(* Logix 5000 project; controller ABB_Drive_Test vendor 1 type 14 code 149 rev 33.12; software revision 33.01; part 2 of 6 *)

        [6600] := 57, [6601] := 46, [6602] := 48, [6603] := 48, [6604] := 48, [6605] := 48, [6606] := 48, [6607] := 48, [6608] := 48, [6609] := 48, [6610] := 44, [6611] := 49, [6612] := 48, [6613] := 46, [6614] := 48, [6615] := 48, [6616] := 48, [6617] := 48, [6618] := 48, [6619] := 48, [6620] := 48, [6621] := 44, [6622] := 49, [6623] := 49, [6624] := 46, [6625] := 48, [6626] := 48, [6627] := 48, [6628] := 48, [6629] := 48, [6630] := 48, [6631] := 48, [6632] := 44, [6633] := 49, [6634] := 50, [6635] := 46, [6636] := 48, [6637] := 48, [6638] := 48, [6639] := 48, [6640] := 48, [6641] := 48, [6642] := 48, [6643] := 44, [6644] := 49, [6645] := 46, [6646] := 48, [6647] := 48, [6648] := 48, [6649] := 48, [6650] := 48, [6651] := 48, [6652] := 48, [6653] := 48, [6654] := 13, [6655] := 10, [6656] := 51, [6657] := 53, [6658] := 56, [6659] := 56,
        [6660] := 56, [6661] := 44, [6662] := 48, [6663] := 46, [6664] := 48, [6665] := 57, [6666] := 51, [6667] := 51, [6668] := 48, [6669] := 56, [6670] := 52, [6671] := 54, [6672] := 44, [6673] := 50, [6674] := 46, [6675] := 48, [6676] := 48, [6677] := 48, [6678] := 48, [6679] := 48, [6680] := 48, [6681] := 48, [6682] := 48, [6683] := 44, [6684] := 53, [6685] := 46, [6686] := 48, [6687] := 48, [6688] := 48, [6689] := 48, [6690] := 48, [6691] := 48, [6692] := 48, [6693] := 48, [6694] := 44, [6695] := 54, [6696] := 46, [6697] := 48, [6698] := 48, [6699] := 48, [6700] := 48, [6701] := 48, [6702] := 48, [6703] := 48, [6704] := 48, [6705] := 44, [6706] := 55, [6707] := 46, [6708] := 48, [6709] := 48, [6710] := 48, [6711] := 48, [6712] := 48, [6713] := 48, [6714] := 48, [6715] := 48, [6716] := 44, [6717] := 56, [6718] := 46, [6719] := 48,
        [6720] := 48, [6721] := 48, [6722] := 48, [6723] := 48, [6724] := 48, [6725] := 48, [6726] := 48, [6727] := 44, [6728] := 57, [6729] := 46, [6730] := 48, [6731] := 48, [6732] := 48, [6733] := 48, [6734] := 48, [6735] := 48, [6736] := 48, [6737] := 48, [6738] := 44, [6739] := 49, [6740] := 48, [6741] := 46, [6742] := 48, [6743] := 48, [6744] := 48, [6745] := 48, [6746] := 48, [6747] := 48, [6748] := 48, [6749] := 44, [6750] := 49, [6751] := 49, [6752] := 46, [6753] := 48, [6754] := 48, [6755] := 48, [6756] := 48, [6757] := 48, [6758] := 48, [6759] := 48, [6760] := 44, [6761] := 49, [6762] := 50, [6763] := 46, [6764] := 48, [6765] := 48, [6766] := 48, [6767] := 48, [6768] := 48, [6769] := 48, [6770] := 48, [6771] := 44, [6772] := 49, [6773] := 46, [6774] := 48, [6775] := 48, [6776] := 48, [6777] := 48, [6778] := 48, [6779] := 48,
        [6780] := 48, [6781] := 48, [6782] := 13, [6783] := 10, [6784] := 51, [6785] := 53, [6786] := 56, [6787] := 56, [6788] := 56, [6789] := 44, [6790] := 48, [6791] := 46, [6792] := 48, [6793] := 57, [6794] := 51, [6795] := 51, [6796] := 50, [6797] := 48, [6798] := 48, [6799] := 50, [6800] := 44, [6801] := 50, [6802] := 46, [6803] := 48, [6804] := 48, [6805] := 48, [6806] := 48, [6807] := 48, [6808] := 48, [6809] := 48, [6810] := 48, [6811] := 44, [6812] := 53, [6813] := 46, [6814] := 48, [6815] := 48, [6816] := 48, [6817] := 48, [6818] := 48, [6819] := 48, [6820] := 48, [6821] := 48, [6822] := 44, [6823] := 54, [6824] := 46, [6825] := 48, [6826] := 48, [6827] := 48, [6828] := 48, [6829] := 48, [6830] := 48, [6831] := 48, [6832] := 48, [6833] := 44, [6834] := 55, [6835] := 46, [6836] := 48, [6837] := 48, [6838] := 48, [6839] := 48,
        [6840] := 48, [6841] := 48, [6842] := 48, [6843] := 48, [6844] := 44, [6845] := 56, [6846] := 46, [6847] := 48, [6848] := 48, [6849] := 48, [6850] := 48, [6851] := 48, [6852] := 48, [6853] := 48, [6854] := 48, [6855] := 44, [6856] := 57, [6857] := 46, [6858] := 48, [6859] := 48, [6860] := 48, [6861] := 48, [6862] := 48, [6863] := 48, [6864] := 48, [6865] := 48, [6866] := 44, [6867] := 49, [6868] := 48, [6869] := 46, [6870] := 48, [6871] := 48, [6872] := 48, [6873] := 48, [6874] := 48, [6875] := 48, [6876] := 48, [6877] := 44, [6878] := 49, [6879] := 49, [6880] := 46, [6881] := 48, [6882] := 48, [6883] := 48, [6884] := 48, [6885] := 48, [6886] := 48, [6887] := 48, [6888] := 44, [6889] := 49, [6890] := 50, [6891] := 46, [6892] := 48, [6893] := 48, [6894] := 48, [6895] := 48, [6896] := 48, [6897] := 48, [6898] := 48, [6899] := 44,
        [6900] := 49, [6901] := 46, [6902] := 48, [6903] := 48, [6904] := 48, [6905] := 48, [6906] := 48, [6907] := 48, [6908] := 48, [6909] := 48, [6910] := 13, [6911] := 10, [6912] := 51, [6913] := 53, [6914] := 56, [6915] := 56, [6916] := 56, [6917] := 44, [6918] := 48, [6919] := 46, [6920] := 48, [6921] := 57, [6922] := 51, [6923] := 51, [6924] := 51, [6925] := 49, [6926] := 54, [6927] := 48, [6928] := 44, [6929] := 50, [6930] := 46, [6931] := 48, [6932] := 48, [6933] := 48, [6934] := 48, [6935] := 48, [6936] := 48, [6937] := 48, [6938] := 48, [6939] := 44, [6940] := 53, [6941] := 46, [6942] := 48, [6943] := 48, [6944] := 48, [6945] := 48, [6946] := 48, [6947] := 48, [6948] := 48, [6949] := 48, [6950] := 44, [6951] := 54, [6952] := 46, [6953] := 48, [6954] := 48, [6955] := 48, [6956] := 48, [6957] := 48, [6958] := 48, [6959] := 48,
        [6960] := 48, [6961] := 44, [6962] := 55, [6963] := 46, [6964] := 48, [6965] := 48, [6966] := 48, [6967] := 48, [6968] := 48, [6969] := 48, [6970] := 48, [6971] := 48, [6972] := 44, [6973] := 56, [6974] := 46, [6975] := 48, [6976] := 48, [6977] := 48, [6978] := 48, [6979] := 48, [6980] := 48, [6981] := 48, [6982] := 48, [6983] := 44, [6984] := 57, [6985] := 46, [6986] := 48, [6987] := 48, [6988] := 48, [6989] := 48, [6990] := 48, [6991] := 48, [6992] := 48, [6993] := 48, [6994] := 44, [6995] := 49, [6996] := 48, [6997] := 46, [6998] := 48, [6999] := 48, [7000] := 48, [7001] := 48, [7002] := 48, [7003] := 48, [7004] := 48, [7005] := 44, [7006] := 49, [7007] := 49, [7008] := 46, [7009] := 48, [7010] := 48, [7011] := 48, [7012] := 48, [7013] := 48, [7014] := 48, [7015] := 48, [7016] := 44, [7017] := 49, [7018] := 50, [7019] := 46,
        [7020] := 48, [7021] := 48, [7022] := 48, [7023] := 48, [7024] := 48, [7025] := 48, [7026] := 48, [7027] := 44, [7028] := 49, [7029] := 46, [7030] := 48, [7031] := 48, [7032] := 48, [7033] := 48, [7034] := 48, [7035] := 48, [7036] := 48, [7037] := 48, [7038] := 13, [7039] := 10, [7040] := 51, [7041] := 53, [7042] := 56, [7043] := 56, [7044] := 56, [7045] := 44, [7046] := 48, [7047] := 46, [7048] := 48, [7049] := 57, [7050] := 51, [7051] := 51, [7052] := 52, [7053] := 51, [7054] := 49, [7055] := 55, [7056] := 44, [7057] := 50, [7058] := 46, [7059] := 48, [7060] := 48, [7061] := 48, [7062] := 48, [7063] := 48, [7064] := 48, [7065] := 48, [7066] := 48, [7067] := 44, [7068] := 53, [7069] := 46, [7070] := 48, [7071] := 48, [7072] := 48, [7073] := 48, [7074] := 48, [7075] := 48, [7076] := 48, [7077] := 48, [7078] := 44, [7079] := 54,
        [7080] := 46, [7081] := 48, [7082] := 48, [7083] := 48, [7084] := 48, [7085] := 48, [7086] := 48, [7087] := 48, [7088] := 48, [7089] := 44, [7090] := 55, [7091] := 46, [7092] := 48, [7093] := 48, [7094] := 48, [7095] := 48, [7096] := 48, [7097] := 48, [7098] := 48, [7099] := 48, [7100] := 44, [7101] := 56, [7102] := 46, [7103] := 48, [7104] := 48, [7105] := 48, [7106] := 48, [7107] := 48, [7108] := 48, [7109] := 48, [7110] := 48, [7111] := 44, [7112] := 57, [7113] := 46, [7114] := 48, [7115] := 48, [7116] := 48, [7117] := 48, [7118] := 48, [7119] := 48, [7120] := 48, [7121] := 48, [7122] := 44, [7123] := 49, [7124] := 48, [7125] := 46, [7126] := 48, [7127] := 48, [7128] := 48, [7129] := 48, [7130] := 48, [7131] := 48, [7132] := 48, [7133] := 44, [7134] := 49, [7135] := 49, [7136] := 46, [7137] := 48, [7138] := 48, [7139] := 48,
        [7140] := 48, [7141] := 48, [7142] := 48, [7143] := 48, [7144] := 44, [7145] := 49, [7146] := 50, [7147] := 46, [7148] := 48, [7149] := 48, [7150] := 48, [7151] := 48, [7152] := 48, [7153] := 48, [7154] := 48, [7155] := 44, [7156] := 49, [7157] := 46, [7158] := 48, [7159] := 48, [7160] := 48, [7161] := 48, [7162] := 48, [7163] := 48, [7164] := 48, [7165] := 48, [7166] := 13, [7167] := 10, [7168] := 51, [7169] := 53, [7170] := 56, [7171] := 56, [7172] := 56, [7173] := 44, [7174] := 48, [7175] := 46, [7176] := 48, [7177] := 57, [7178] := 51, [7179] := 51, [7180] := 53, [7181] := 52, [7182] := 55, [7183] := 53, [7184] := 44, [7185] := 50, [7186] := 46, [7187] := 48, [7188] := 48, [7189] := 48, [7190] := 48, [7191] := 48, [7192] := 48, [7193] := 48, [7194] := 48, [7195] := 44, [7196] := 53, [7197] := 46, [7198] := 48, [7199] := 48,
        [7200] := 48, [7201] := 48, [7202] := 48, [7203] := 48, [7204] := 48, [7205] := 48, [7206] := 44, [7207] := 54, [7208] := 46, [7209] := 48, [7210] := 48, [7211] := 48, [7212] := 48, [7213] := 48, [7214] := 48, [7215] := 48, [7216] := 48, [7217] := 44, [7218] := 55, [7219] := 46, [7220] := 48, [7221] := 48, [7222] := 48, [7223] := 48, [7224] := 48, [7225] := 48, [7226] := 48, [7227] := 48, [7228] := 44, [7229] := 56, [7230] := 46, [7231] := 48, [7232] := 48, [7233] := 48, [7234] := 48, [7235] := 48, [7236] := 48, [7237] := 48, [7238] := 48, [7239] := 44, [7240] := 57, [7241] := 46, [7242] := 48, [7243] := 48, [7244] := 48, [7245] := 48, [7246] := 48, [7247] := 48, [7248] := 48, [7249] := 48, [7250] := 44, [7251] := 49, [7252] := 48, [7253] := 46, [7254] := 48, [7255] := 48, [7256] := 48, [7257] := 48, [7258] := 48, [7259] := 48,
        [7260] := 48, [7261] := 44, [7262] := 49, [7263] := 49, [7264] := 46, [7265] := 48, [7266] := 48, [7267] := 48, [7268] := 48, [7269] := 48, [7270] := 48, [7271] := 48, [7272] := 44, [7273] := 49, [7274] := 50, [7275] := 46, [7276] := 48, [7277] := 48, [7278] := 48, [7279] := 48, [7280] := 48, [7281] := 48, [7282] := 48, [7283] := 44, [7284] := 49, [7285] := 46, [7286] := 48, [7287] := 48, [7288] := 48, [7289] := 48, [7290] := 48, [7291] := 48, [7292] := 48, [7293] := 48, [7294] := 13, [7295] := 10, [7296] := 51, [7297] := 53, [7298] := 56, [7299] := 56, [7300] := 56, [7301] := 44, [7302] := 48, [7303] := 46, [7304] := 48, [7305] := 57, [7306] := 51, [7307] := 51, [7308] := 54, [7309] := 54, [7310] := 51, [7311] := 50, [7312] := 44, [7313] := 50, [7314] := 46, [7315] := 48, [7316] := 48, [7317] := 48, [7318] := 48, [7319] := 48,
        [7320] := 48, [7321] := 48, [7322] := 48, [7323] := 44, [7324] := 53, [7325] := 46, [7326] := 48, [7327] := 48, [7328] := 48, [7329] := 48, [7330] := 48, [7331] := 48, [7332] := 48, [7333] := 48, [7334] := 44, [7335] := 54, [7336] := 46, [7337] := 48, [7338] := 48, [7339] := 48, [7340] := 48, [7341] := 48, [7342] := 48, [7343] := 48, [7344] := 48, [7345] := 44, [7346] := 55, [7347] := 46, [7348] := 48, [7349] := 48, [7350] := 48, [7351] := 48, [7352] := 48, [7353] := 48, [7354] := 48, [7355] := 48, [7356] := 44, [7357] := 56, [7358] := 46, [7359] := 48, [7360] := 48, [7361] := 48, [7362] := 48, [7363] := 48, [7364] := 48, [7365] := 48, [7366] := 48, [7367] := 44, [7368] := 57, [7369] := 46, [7370] := 48, [7371] := 48, [7372] := 48, [7373] := 48, [7374] := 48, [7375] := 48, [7376] := 48, [7377] := 48, [7378] := 44, [7379] := 49,
        [7380] := 48, [7381] := 46, [7382] := 48, [7383] := 48, [7384] := 48, [7385] := 48, [7386] := 48, [7387] := 48, [7388] := 48, [7389] := 44, [7390] := 49, [7391] := 49, [7392] := 46, [7393] := 48, [7394] := 48, [7395] := 48, [7396] := 48, [7397] := 48, [7398] := 48, [7399] := 48, [7400] := 44, [7401] := 49, [7402] := 50, [7403] := 46, [7404] := 48, [7405] := 48, [7406] := 48, [7407] := 48, [7408] := 48, [7409] := 48, [7410] := 48, [7411] := 44, [7412] := 49, [7413] := 46, [7414] := 48, [7415] := 48, [7416] := 48, [7417] := 48, [7418] := 48, [7419] := 48, [7420] := 48, [7421] := 48, [7422] := 13, [7423] := 10, [7424] := 51, [7425] := 53, [7426] := 56, [7427] := 56, [7428] := 56, [7429] := 44, [7430] := 48, [7431] := 46, [7432] := 48, [7433] := 57, [7434] := 51, [7435] := 51, [7436] := 55, [7437] := 55, [7438] := 57, [7439] := 48,
        [7440] := 44, [7441] := 50, [7442] := 46, [7443] := 48, [7444] := 48, [7445] := 48, [7446] := 48, [7447] := 48, [7448] := 48, [7449] := 48, [7450] := 48, [7451] := 44, [7452] := 53, [7453] := 46, [7454] := 48, [7455] := 48, [7456] := 48, [7457] := 48, [7458] := 48, [7459] := 48, [7460] := 48, [7461] := 48, [7462] := 44, [7463] := 54, [7464] := 46, [7465] := 48, [7466] := 48, [7467] := 48, [7468] := 48, [7469] := 48, [7470] := 48, [7471] := 48, [7472] := 48, [7473] := 44, [7474] := 55, [7475] := 46, [7476] := 48, [7477] := 48, [7478] := 48, [7479] := 48, [7480] := 48, [7481] := 48, [7482] := 48, [7483] := 48, [7484] := 44, [7485] := 56, [7486] := 46, [7487] := 48, [7488] := 48, [7489] := 48, [7490] := 48, [7491] := 48, [7492] := 48, [7493] := 48, [7494] := 48, [7495] := 44, [7496] := 57, [7497] := 46, [7498] := 48, [7499] := 48,
        [7500] := 48, [7501] := 48, [7502] := 48, [7503] := 48, [7504] := 48, [7505] := 48, [7506] := 44, [7507] := 49, [7508] := 48, [7509] := 46, [7510] := 48, [7511] := 48, [7512] := 48, [7513] := 48, [7514] := 48, [7515] := 48, [7516] := 48, [7517] := 44, [7518] := 49, [7519] := 49, [7520] := 46, [7521] := 48, [7522] := 48, [7523] := 48, [7524] := 48, [7525] := 48, [7526] := 48, [7527] := 48, [7528] := 44, [7529] := 49, [7530] := 50, [7531] := 46, [7532] := 48, [7533] := 48, [7534] := 48, [7535] := 48, [7536] := 48, [7537] := 48, [7538] := 48, [7539] := 44, [7540] := 49, [7541] := 46, [7542] := 48, [7543] := 48, [7544] := 48, [7545] := 48, [7546] := 48, [7547] := 48, [7548] := 48, [7549] := 48, [7550] := 13, [7551] := 10, [7552] := 51, [7553] := 53, [7554] := 56, [7555] := 56, [7556] := 56, [7557] := 44, [7558] := 48, [7559] := 46,
        [7560] := 48, [7561] := 57, [7562] := 51, [7563] := 51, [7564] := 56, [7565] := 57, [7566] := 52, [7567] := 55, [7568] := 44, [7569] := 50, [7570] := 46, [7571] := 48, [7572] := 48, [7573] := 48, [7574] := 48, [7575] := 48, [7576] := 48, [7577] := 48, [7578] := 48, [7579] := 44, [7580] := 53, [7581] := 46, [7582] := 48, [7583] := 48, [7584] := 48, [7585] := 48, [7586] := 48, [7587] := 48, [7588] := 48, [7589] := 48, [7590] := 44, [7591] := 54, [7592] := 46, [7593] := 48, [7594] := 48, [7595] := 48, [7596] := 48, [7597] := 48, [7598] := 48, [7599] := 48, [7600] := 48, [7601] := 44, [7602] := 55, [7603] := 46, [7604] := 48, [7605] := 48, [7606] := 48, [7607] := 48, [7608] := 48, [7609] := 48, [7610] := 48, [7611] := 48, [7612] := 44, [7613] := 56, [7614] := 46, [7615] := 48, [7616] := 48, [7617] := 48, [7618] := 48, [7619] := 48,
        [7620] := 48, [7621] := 48, [7622] := 48, [7623] := 44, [7624] := 57, [7625] := 46, [7626] := 48, [7627] := 48, [7628] := 48, [7629] := 48, [7630] := 48, [7631] := 48, [7632] := 48, [7633] := 48, [7634] := 44, [7635] := 49, [7636] := 48, [7637] := 46, [7638] := 48, [7639] := 48, [7640] := 48, [7641] := 48, [7642] := 48, [7643] := 48, [7644] := 48, [7645] := 44, [7646] := 49, [7647] := 49, [7648] := 46, [7649] := 48, [7650] := 48, [7651] := 48, [7652] := 48, [7653] := 48, [7654] := 48, [7655] := 48, [7656] := 44, [7657] := 49, [7658] := 50, [7659] := 46, [7660] := 48, [7661] := 48, [7662] := 48, [7663] := 48, [7664] := 48, [7665] := 48, [7666] := 48, [7667] := 44, [7668] := 49, [7669] := 46, [7670] := 48, [7671] := 48, [7672] := 48, [7673] := 48, [7674] := 48, [7675] := 48, [7676] := 48, [7677] := 48, [7678] := 13, [7679] := 10,
        [7680] := 51, [7681] := 53, [7682] := 56, [7683] := 56, [7684] := 56, [7685] := 44, [7686] := 48, [7687] := 46, [7688] := 48, [7689] := 57, [7690] := 51, [7691] := 52, [7692] := 48, [7693] := 49, [7694] := 48, [7695] := 52, [7696] := 44, [7697] := 50, [7698] := 46, [7699] := 48, [7700] := 48, [7701] := 48, [7702] := 48, [7703] := 48, [7704] := 48, [7705] := 48, [7706] := 48, [7707] := 44, [7708] := 53, [7709] := 46, [7710] := 48, [7711] := 48, [7712] := 48, [7713] := 48, [7714] := 48, [7715] := 48, [7716] := 48, [7717] := 48, [7718] := 44, [7719] := 54, [7720] := 46, [7721] := 48, [7722] := 48, [7723] := 48, [7724] := 48, [7725] := 48, [7726] := 48, [7727] := 48, [7728] := 48, [7729] := 44, [7730] := 55, [7731] := 46, [7732] := 48, [7733] := 48, [7734] := 48, [7735] := 48, [7736] := 48, [7737] := 48, [7738] := 48, [7739] := 48,
        [7740] := 44, [7741] := 56, [7742] := 46, [7743] := 48, [7744] := 48, [7745] := 48, [7746] := 48, [7747] := 48, [7748] := 48, [7749] := 48, [7750] := 48, [7751] := 44, [7752] := 57, [7753] := 46, [7754] := 48, [7755] := 48, [7756] := 48, [7757] := 48, [7758] := 48, [7759] := 48, [7760] := 48, [7761] := 48, [7762] := 44, [7763] := 49, [7764] := 48, [7765] := 46, [7766] := 48, [7767] := 48, [7768] := 48, [7769] := 48, [7770] := 48, [7771] := 48, [7772] := 48, [7773] := 44, [7774] := 49, [7775] := 49, [7776] := 46, [7777] := 48, [7778] := 48, [7779] := 48, [7780] := 48, [7781] := 48, [7782] := 48, [7783] := 48, [7784] := 44, [7785] := 49, [7786] := 50, [7787] := 46, [7788] := 48, [7789] := 48, [7790] := 48, [7791] := 48, [7792] := 48, [7793] := 48, [7794] := 48, [7795] := 44, [7796] := 49, [7797] := 46, [7798] := 48, [7799] := 48,
        [7800] := 48, [7801] := 48, [7802] := 48, [7803] := 48, [7804] := 48, [7805] := 48, [7806] := 13, [7807] := 10, [7808] := 51, [7809] := 53, [7810] := 56, [7811] := 56, [7812] := 56, [7813] := 44, [7814] := 48, [7815] := 46, [7816] := 48, [7817] := 57, [7818] := 51, [7819] := 52, [7820] := 49, [7821] := 50, [7822] := 54, [7823] := 50, [7824] := 44, [7825] := 50, [7826] := 46, [7827] := 48, [7828] := 48, [7829] := 48, [7830] := 48, [7831] := 48, [7832] := 48, [7833] := 48, [7834] := 48, [7835] := 44, [7836] := 53, [7837] := 46, [7838] := 48, [7839] := 48, [7840] := 48, [7841] := 48, [7842] := 48, [7843] := 48, [7844] := 48, [7845] := 48, [7846] := 44, [7847] := 54, [7848] := 46, [7849] := 48, [7850] := 48, [7851] := 48, [7852] := 48, [7853] := 48, [7854] := 48, [7855] := 48, [7856] := 48, [7857] := 44, [7858] := 55, [7859] := 46,
        [7860] := 48, [7861] := 48, [7862] := 48, [7863] := 48, [7864] := 48, [7865] := 48, [7866] := 48, [7867] := 48, [7868] := 44, [7869] := 56, [7870] := 46, [7871] := 48, [7872] := 48, [7873] := 48, [7874] := 48, [7875] := 48, [7876] := 48, [7877] := 48, [7878] := 48, [7879] := 44, [7880] := 57, [7881] := 46, [7882] := 48, [7883] := 48, [7884] := 48, [7885] := 48, [7886] := 48, [7887] := 48, [7888] := 48, [7889] := 48, [7890] := 44, [7891] := 49, [7892] := 48, [7893] := 46, [7894] := 48, [7895] := 48, [7896] := 48, [7897] := 48, [7898] := 48, [7899] := 48, [7900] := 48, [7901] := 44, [7902] := 49, [7903] := 49, [7904] := 46, [7905] := 48, [7906] := 48, [7907] := 48, [7908] := 48, [7909] := 48, [7910] := 48, [7911] := 48, [7912] := 44, [7913] := 49, [7914] := 50, [7915] := 46, [7916] := 48, [7917] := 48, [7918] := 48, [7919] := 48,
        [7920] := 48, [7921] := 48, [7922] := 48, [7923] := 44, [7924] := 49, [7925] := 46, [7926] := 48, [7927] := 48, [7928] := 48, [7929] := 48, [7930] := 48, [7931] := 48, [7932] := 48, [7933] := 48, [7934] := 13, [7935] := 10, [7936] := 51, [7937] := 53, [7938] := 56, [7939] := 56, [7940] := 56, [7941] := 44, [7942] := 48, [7943] := 46, [7944] := 48, [7945] := 57, [7946] := 51, [7947] := 52, [7948] := 50, [7949] := 52, [7950] := 49, [7951] := 57, [7952] := 44, [7953] := 50, [7954] := 46, [7955] := 48, [7956] := 48, [7957] := 48, [7958] := 48, [7959] := 48, [7960] := 48, [7961] := 48, [7962] := 48, [7963] := 44, [7964] := 53, [7965] := 46, [7966] := 48, [7967] := 48, [7968] := 48, [7969] := 48, [7970] := 48, [7971] := 48, [7972] := 48, [7973] := 48, [7974] := 44, [7975] := 54, [7976] := 46, [7977] := 48, [7978] := 48, [7979] := 48,
        [7980] := 48, [7981] := 48, [7982] := 48, [7983] := 48, [7984] := 48, [7985] := 44, [7986] := 55, [7987] := 46, [7988] := 48, [7989] := 48, [7990] := 48, [7991] := 48, [7992] := 48, [7993] := 48, [7994] := 48, [7995] := 48, [7996] := 44, [7997] := 56, [7998] := 46, [7999] := 48, [8000] := 48, [8001] := 48, [8002] := 48, [8003] := 48, [8004] := 48, [8005] := 48, [8006] := 48, [8007] := 44, [8008] := 57, [8009] := 46, [8010] := 48, [8011] := 48, [8012] := 48, [8013] := 48, [8014] := 48, [8015] := 48, [8016] := 48, [8017] := 48, [8018] := 44, [8019] := 49, [8020] := 48, [8021] := 46, [8022] := 48, [8023] := 48, [8024] := 48, [8025] := 48, [8026] := 48, [8027] := 48, [8028] := 48, [8029] := 44, [8030] := 49, [8031] := 49, [8032] := 46, [8033] := 48, [8034] := 48, [8035] := 48, [8036] := 48, [8037] := 48, [8038] := 48, [8039] := 48,
        [8040] := 44, [8041] := 49, [8042] := 50, [8043] := 46, [8044] := 48, [8045] := 48, [8046] := 48, [8047] := 48, [8048] := 48, [8049] := 48, [8050] := 48, [8051] := 44, [8052] := 49, [8053] := 46, [8054] := 48, [8055] := 48, [8056] := 48, [8057] := 48, [8058] := 48, [8059] := 48, [8060] := 48, [8061] := 48, [8062] := 13, [8063] := 10, [8064] := 51, [8065] := 53, [8066] := 56, [8067] := 56, [8068] := 56, [8069] := 44, [8070] := 48, [8071] := 46, [8072] := 48, [8073] := 57, [8074] := 51, [8075] := 52, [8076] := 51, [8077] := 53, [8078] := 55, [8079] := 55, [8080] := 44, [8081] := 50, [8082] := 46, [8083] := 48, [8084] := 48, [8085] := 48, [8086] := 48, [8087] := 48, [8088] := 48, [8089] := 48, [8090] := 48, [8091] := 44, [8092] := 53, [8093] := 46, [8094] := 48, [8095] := 48, [8096] := 48, [8097] := 48, [8098] := 48, [8099] := 48,
        [8100] := 48, [8101] := 48, [8102] := 44, [8103] := 54, [8104] := 46, [8105] := 48, [8106] := 48, [8107] := 48, [8108] := 48, [8109] := 48, [8110] := 48, [8111] := 48, [8112] := 48, [8113] := 44, [8114] := 55, [8115] := 46, [8116] := 48, [8117] := 48, [8118] := 48, [8119] := 48, [8120] := 48, [8121] := 48, [8122] := 48, [8123] := 48, [8124] := 44, [8125] := 56, [8126] := 46, [8127] := 48, [8128] := 48, [8129] := 48, [8130] := 48, [8131] := 48, [8132] := 48, [8133] := 48, [8134] := 48, [8135] := 44, [8136] := 57, [8137] := 46, [8138] := 48, [8139] := 48, [8140] := 48, [8141] := 48, [8142] := 48, [8143] := 48, [8144] := 48, [8145] := 48, [8146] := 44, [8147] := 49, [8148] := 48, [8149] := 46, [8150] := 48, [8151] := 48, [8152] := 48, [8153] := 48, [8154] := 48, [8155] := 48, [8156] := 48, [8157] := 44, [8158] := 49, [8159] := 49,
        [8160] := 46, [8161] := 48, [8162] := 48, [8163] := 48, [8164] := 48, [8165] := 48, [8166] := 48, [8167] := 48, [8168] := 44, [8169] := 49, [8170] := 50, [8171] := 46, [8172] := 48, [8173] := 48, [8174] := 48, [8175] := 48, [8176] := 48, [8177] := 48, [8178] := 48, [8179] := 44, [8180] := 49, [8181] := 46, [8182] := 48, [8183] := 48, [8184] := 48, [8185] := 48, [8186] := 48, [8187] := 48, [8188] := 48, [8189] := 48, [8190] := 13, [8191] := 10, [8192] := 51, [8193] := 53, [8194] := 56, [8195] := 56, [8196] := 56, [8197] := 44, [8198] := 48, [8199] := 46, [8200] := 48, [8201] := 57, [8202] := 51, [8203] := 52, [8204] := 52, [8205] := 55, [8206] := 51, [8207] := 52, [8208] := 44, [8209] := 50, [8210] := 46, [8211] := 48, [8212] := 48, [8213] := 48, [8214] := 48, [8215] := 48, [8216] := 48, [8217] := 48, [8218] := 48, [8219] := 44,
        [8220] := 53, [8221] := 46, [8222] := 48, [8223] := 48, [8224] := 48, [8225] := 48, [8226] := 48, [8227] := 48, [8228] := 48, [8229] := 48, [8230] := 44, [8231] := 54, [8232] := 46, [8233] := 48, [8234] := 48, [8235] := 48, [8236] := 48, [8237] := 48, [8238] := 48, [8239] := 48, [8240] := 48, [8241] := 44, [8242] := 55, [8243] := 46, [8244] := 48, [8245] := 48, [8246] := 48, [8247] := 48, [8248] := 48, [8249] := 48, [8250] := 48, [8251] := 48, [8252] := 44, [8253] := 56, [8254] := 46, [8255] := 48, [8256] := 48, [8257] := 48, [8258] := 48, [8259] := 48, [8260] := 48, [8261] := 48, [8262] := 48, [8263] := 44, [8264] := 57, [8265] := 46, [8266] := 48, [8267] := 48, [8268] := 48, [8269] := 48, [8270] := 48, [8271] := 48, [8272] := 48, [8273] := 48, [8274] := 44, [8275] := 49, [8276] := 48, [8277] := 46, [8278] := 48, [8279] := 48,
        [8280] := 48, [8281] := 48, [8282] := 48, [8283] := 48, [8284] := 48, [8285] := 44, [8286] := 49, [8287] := 49, [8288] := 46, [8289] := 48, [8290] := 48, [8291] := 48, [8292] := 48, [8293] := 48, [8294] := 48, [8295] := 48, [8296] := 44, [8297] := 49, [8298] := 50, [8299] := 46, [8300] := 48, [8301] := 48, [8302] := 48, [8303] := 48, [8304] := 48, [8305] := 48, [8306] := 48, [8307] := 44, [8308] := 49, [8309] := 46, [8310] := 48, [8311] := 48, [8312] := 48, [8313] := 48, [8314] := 48, [8315] := 48, [8316] := 48, [8317] := 48, [8318] := 13, [8319] := 10, [8320] := 51, [8321] := 53, [8322] := 56, [8323] := 56, [8324] := 56, [8325] := 44, [8326] := 48, [8327] := 46, [8328] := 48, [8329] := 57, [8330] := 51, [8331] := 52, [8332] := 53, [8333] := 56, [8334] := 57, [8335] := 50, [8336] := 44, [8337] := 50, [8338] := 46, [8339] := 48,
        [8340] := 48, [8341] := 48, [8342] := 48, [8343] := 48, [8344] := 48, [8345] := 48, [8346] := 48, [8347] := 44, [8348] := 53, [8349] := 46, [8350] := 48, [8351] := 48, [8352] := 48, [8353] := 48, [8354] := 48, [8355] := 48, [8356] := 48, [8357] := 48, [8358] := 44, [8359] := 54, [8360] := 46, [8361] := 48, [8362] := 48, [8363] := 48, [8364] := 48, [8365] := 48, [8366] := 48, [8367] := 48, [8368] := 48, [8369] := 44, [8370] := 55, [8371] := 46, [8372] := 48, [8373] := 48, [8374] := 48, [8375] := 48, [8376] := 48, [8377] := 48, [8378] := 48, [8379] := 48, [8380] := 44, [8381] := 56, [8382] := 46, [8383] := 48, [8384] := 48, [8385] := 48, [8386] := 48, [8387] := 48, [8388] := 48, [8389] := 48, [8390] := 48, [8391] := 44, [8392] := 57, [8393] := 46, [8394] := 48, [8395] := 48, [8396] := 48, [8397] := 48, [8398] := 48, [8399] := 48,
        [8400] := 48, [8401] := 48, [8402] := 44, [8403] := 49, [8404] := 48, [8405] := 46, [8406] := 48, [8407] := 48, [8408] := 48, [8409] := 48, [8410] := 48, [8411] := 48, [8412] := 48, [8413] := 44, [8414] := 49, [8415] := 49, [8416] := 46, [8417] := 48, [8418] := 48, [8419] := 48, [8420] := 48, [8421] := 48, [8422] := 48, [8423] := 48, [8424] := 44, [8425] := 49, [8426] := 50, [8427] := 46, [8428] := 48, [8429] := 48, [8430] := 48, [8431] := 48, [8432] := 48, [8433] := 48, [8434] := 48, [8435] := 44, [8436] := 49, [8437] := 46, [8438] := 48, [8439] := 48, [8440] := 48, [8441] := 48, [8442] := 48, [8443] := 48, [8444] := 48, [8445] := 48, [8446] := 13, [8447] := 10, [8448] := 51, [8449] := 53, [8450] := 56, [8451] := 56, [8452] := 56, [8453] := 44, [8454] := 48, [8455] := 46, [8456] := 48, [8457] := 57, [8458] := 51, [8459] := 52,
        [8460] := 55, [8461] := 48, [8462] := 52, [8463] := 57, [8464] := 44, [8465] := 50, [8466] := 46, [8467] := 48, [8468] := 48, [8469] := 48, [8470] := 48, [8471] := 48, [8472] := 48, [8473] := 48, [8474] := 48, [8475] := 44, [8476] := 53, [8477] := 46, [8478] := 48, [8479] := 48, [8480] := 48, [8481] := 48, [8482] := 48, [8483] := 48, [8484] := 48, [8485] := 48, [8486] := 44, [8487] := 54, [8488] := 46, [8489] := 48, [8490] := 48, [8491] := 48, [8492] := 48, [8493] := 48, [8494] := 48, [8495] := 48, [8496] := 48, [8497] := 44, [8498] := 55, [8499] := 46, [8500] := 48, [8501] := 48, [8502] := 48, [8503] := 48, [8504] := 48, [8505] := 48, [8506] := 48, [8507] := 48, [8508] := 44, [8509] := 56, [8510] := 46, [8511] := 48, [8512] := 48, [8513] := 48, [8514] := 48, [8515] := 48, [8516] := 48, [8517] := 48, [8518] := 48, [8519] := 44,
        [8520] := 57, [8521] := 46, [8522] := 48, [8523] := 48, [8524] := 48, [8525] := 48, [8526] := 48, [8527] := 48, [8528] := 48, [8529] := 48, [8530] := 44, [8531] := 49, [8532] := 48, [8533] := 46, [8534] := 48, [8535] := 48, [8536] := 48, [8537] := 48, [8538] := 48, [8539] := 48, [8540] := 48, [8541] := 44, [8542] := 49, [8543] := 49, [8544] := 46, [8545] := 48, [8546] := 48, [8547] := 48, [8548] := 48, [8549] := 48, [8550] := 48, [8551] := 48, [8552] := 44, [8553] := 49, [8554] := 50, [8555] := 46, [8556] := 48, [8557] := 48, [8558] := 48, [8559] := 48, [8560] := 48, [8561] := 48, [8562] := 48, [8563] := 44, [8564] := 49, [8565] := 46, [8566] := 48, [8567] := 48, [8568] := 48, [8569] := 48, [8570] := 48, [8571] := 48, [8572] := 48, [8573] := 48, [8574] := 13, [8575] := 10, [8576] := 51, [8577] := 53, [8578] := 56, [8579] := 56,
        [8580] := 56, [8581] := 44, [8582] := 48, [8583] := 46, [8584] := 48, [8585] := 57, [8586] := 51, [8587] := 52, [8588] := 56, [8589] := 50, [8590] := 48, [8591] := 55, [8592] := 44, [8593] := 50, [8594] := 46, [8595] := 48, [8596] := 48, [8597] := 48, [8598] := 48, [8599] := 48, [8600] := 48, [8601] := 48, [8602] := 48, [8603] := 44, [8604] := 53, [8605] := 46, [8606] := 48, [8607] := 48, [8608] := 48, [8609] := 48, [8610] := 48, [8611] := 48, [8612] := 48, [8613] := 48, [8614] := 44, [8615] := 54, [8616] := 46, [8617] := 48, [8618] := 48, [8619] := 48, [8620] := 48, [8621] := 48, [8622] := 48, [8623] := 48, [8624] := 48, [8625] := 44, [8626] := 55, [8627] := 46, [8628] := 48, [8629] := 48, [8630] := 48, [8631] := 48, [8632] := 48, [8633] := 48, [8634] := 48, [8635] := 48, [8636] := 44, [8637] := 56, [8638] := 46, [8639] := 48,
        [8640] := 48, [8641] := 48, [8642] := 48, [8643] := 48, [8644] := 48, [8645] := 48, [8646] := 48, [8647] := 44, [8648] := 57, [8649] := 46, [8650] := 48, [8651] := 48, [8652] := 48, [8653] := 48, [8654] := 48, [8655] := 48, [8656] := 48, [8657] := 48, [8658] := 44, [8659] := 49, [8660] := 48, [8661] := 46, [8662] := 48, [8663] := 48, [8664] := 48, [8665] := 48, [8666] := 48, [8667] := 48, [8668] := 48, [8669] := 44, [8670] := 49, [8671] := 49, [8672] := 46, [8673] := 48, [8674] := 48, [8675] := 48, [8676] := 48, [8677] := 48, [8678] := 48, [8679] := 48, [8680] := 44, [8681] := 49, [8682] := 50, [8683] := 46, [8684] := 48, [8685] := 48, [8686] := 48, [8687] := 48, [8688] := 48, [8689] := 48, [8690] := 48, [8691] := 44, [8692] := 49, [8693] := 46, [8694] := 48, [8695] := 48, [8696] := 48, [8697] := 48, [8698] := 48, [8699] := 48,
        [8700] := 48, [8701] := 48, [8702] := 13, [8703] := 10, [8704] := 51, [8705] := 53, [8706] := 56, [8707] := 56, [8708] := 56, [8709] := 44, [8710] := 48, [8711] := 46, [8712] := 48, [8713] := 57, [8714] := 51, [8715] := 52, [8716] := 57, [8717] := 51, [8718] := 54, [8719] := 51, [8720] := 44, [8721] := 50, [8722] := 46, [8723] := 48, [8724] := 48, [8725] := 48, [8726] := 48, [8727] := 48, [8728] := 48, [8729] := 48, [8730] := 48, [8731] := 44, [8732] := 53, [8733] := 46, [8734] := 48, [8735] := 48, [8736] := 48, [8737] := 48, [8738] := 48, [8739] := 48, [8740] := 48, [8741] := 48, [8742] := 44, [8743] := 54, [8744] := 46, [8745] := 48, [8746] := 48, [8747] := 48, [8748] := 48, [8749] := 48, [8750] := 48, [8751] := 48, [8752] := 48, [8753] := 44, [8754] := 55, [8755] := 46, [8756] := 48, [8757] := 48, [8758] := 48, [8759] := 48,
        [8760] := 48, [8761] := 48, [8762] := 48, [8763] := 48, [8764] := 44, [8765] := 56, [8766] := 46, [8767] := 48, [8768] := 48, [8769] := 48, [8770] := 48, [8771] := 48, [8772] := 48, [8773] := 48, [8774] := 48, [8775] := 44, [8776] := 57, [8777] := 46, [8778] := 48, [8779] := 48, [8780] := 48, [8781] := 48, [8782] := 48, [8783] := 48, [8784] := 48, [8785] := 48, [8786] := 44, [8787] := 49, [8788] := 48, [8789] := 46, [8790] := 48, [8791] := 48, [8792] := 48, [8793] := 48, [8794] := 48, [8795] := 48, [8796] := 48, [8797] := 44, [8798] := 49, [8799] := 49, [8800] := 46, [8801] := 48, [8802] := 48, [8803] := 48, [8804] := 48, [8805] := 48, [8806] := 48, [8807] := 48, [8808] := 44, [8809] := 49, [8810] := 50, [8811] := 46, [8812] := 48, [8813] := 48, [8814] := 48, [8815] := 48, [8816] := 48, [8817] := 48, [8818] := 48, [8819] := 44,
        [8820] := 49, [8821] := 46, [8822] := 48, [8823] := 48, [8824] := 48, [8825] := 48, [8826] := 48, [8827] := 48, [8828] := 48, [8829] := 48, [8830] := 13, [8831] := 10, [8832] := 51, [8833] := 53, [8834] := 56, [8835] := 56, [8836] := 56, [8837] := 44, [8838] := 48, [8839] := 46, [8840] := 48, [8841] := 57, [8842] := 51, [8843] := 53, [8844] := 48, [8845] := 53, [8846] := 50, [8847] := 49, [8848] := 44, [8849] := 50, [8850] := 46, [8851] := 48, [8852] := 48, [8853] := 48, [8854] := 48, [8855] := 48, [8856] := 48, [8857] := 48, [8858] := 48, [8859] := 44, [8860] := 53, [8861] := 46, [8862] := 48, [8863] := 48, [8864] := 48, [8865] := 48, [8866] := 48, [8867] := 48, [8868] := 48, [8869] := 48, [8870] := 44, [8871] := 54, [8872] := 46, [8873] := 48, [8874] := 48, [8875] := 48, [8876] := 48, [8877] := 48, [8878] := 48, [8879] := 48,
        [8880] := 48, [8881] := 44, [8882] := 55, [8883] := 46, [8884] := 48, [8885] := 48, [8886] := 48, [8887] := 48, [8888] := 48, [8889] := 48, [8890] := 48, [8891] := 48, [8892] := 44, [8893] := 56, [8894] := 46, [8895] := 48, [8896] := 48, [8897] := 48, [8898] := 48, [8899] := 48, [8900] := 48, [8901] := 48, [8902] := 48, [8903] := 44, [8904] := 57, [8905] := 46, [8906] := 48, [8907] := 48, [8908] := 48, [8909] := 48, [8910] := 48, [8911] := 48, [8912] := 48, [8913] := 48, [8914] := 44, [8915] := 49, [8916] := 48, [8917] := 46, [8918] := 48, [8919] := 48, [8920] := 48, [8921] := 48, [8922] := 48, [8923] := 48, [8924] := 48, [8925] := 44, [8926] := 49, [8927] := 49, [8928] := 46, [8929] := 48, [8930] := 48, [8931] := 48, [8932] := 48, [8933] := 48, [8934] := 48, [8935] := 48, [8936] := 44, [8937] := 49, [8938] := 50, [8939] := 46,
        [8940] := 48, [8941] := 48, [8942] := 48, [8943] := 48, [8944] := 48, [8945] := 48, [8946] := 48, [8947] := 44, [8948] := 49, [8949] := 46, [8950] := 48, [8951] := 48, [8952] := 48, [8953] := 48, [8954] := 48, [8955] := 48, [8956] := 48, [8957] := 48, [8958] := 13, [8959] := 10, [8960] := 51, [8961] := 53, [8962] := 56, [8963] := 56, [8964] := 56, [8965] := 44, [8966] := 48, [8967] := 46, [8968] := 48, [8969] := 57, [8970] := 51, [8971] := 53, [8972] := 49, [8973] := 54, [8974] := 55, [8975] := 57, [8976] := 44, [8977] := 50, [8978] := 46, [8979] := 48, [8980] := 48, [8981] := 48, [8982] := 48, [8983] := 48, [8984] := 48, [8985] := 48, [8986] := 48, [8987] := 44, [8988] := 53, [8989] := 46, [8990] := 48, [8991] := 48, [8992] := 48, [8993] := 48, [8994] := 48, [8995] := 48, [8996] := 48, [8997] := 48, [8998] := 44, [8999] := 54,
        [9000] := 46, [9001] := 48, [9002] := 48, [9003] := 48, [9004] := 48, [9005] := 48, [9006] := 48, [9007] := 48, [9008] := 48, [9009] := 44, [9010] := 55, [9011] := 46, [9012] := 48, [9013] := 48, [9014] := 48, [9015] := 48, [9016] := 48, [9017] := 48, [9018] := 48, [9019] := 48, [9020] := 44, [9021] := 56, [9022] := 46, [9023] := 48, [9024] := 48, [9025] := 48, [9026] := 48, [9027] := 48, [9028] := 48, [9029] := 48, [9030] := 48, [9031] := 44, [9032] := 57, [9033] := 46, [9034] := 48, [9035] := 48, [9036] := 48, [9037] := 48, [9038] := 48, [9039] := 48, [9040] := 48, [9041] := 48, [9042] := 44, [9043] := 49, [9044] := 48, [9045] := 46, [9046] := 48, [9047] := 48, [9048] := 48, [9049] := 48, [9050] := 48, [9051] := 48, [9052] := 48, [9053] := 44, [9054] := 49, [9055] := 49, [9056] := 46, [9057] := 48, [9058] := 48, [9059] := 48,
        [9060] := 48, [9061] := 48, [9062] := 48, [9063] := 48, [9064] := 44, [9065] := 49, [9066] := 50, [9067] := 46, [9068] := 48, [9069] := 48, [9070] := 48, [9071] := 48, [9072] := 48, [9073] := 48, [9074] := 48, [9075] := 44, [9076] := 49, [9077] := 46, [9078] := 48, [9079] := 48, [9080] := 48, [9081] := 48, [9082] := 48, [9083] := 48, [9084] := 48, [9085] := 48, [9086] := 13, [9087] := 10, [9088] := 51, [9089] := 53, [9090] := 56, [9091] := 56, [9092] := 56, [9093] := 44, [9094] := 48, [9095] := 46, [9096] := 48, [9097] := 57, [9098] := 51, [9099] := 53, [9100] := 50, [9101] := 56, [9102] := 51, [9103] := 54, [9104] := 44, [9105] := 50, [9106] := 46, [9107] := 48, [9108] := 48, [9109] := 48, [9110] := 48, [9111] := 48, [9112] := 48, [9113] := 48, [9114] := 48, [9115] := 44, [9116] := 53, [9117] := 46, [9118] := 48, [9119] := 48,
        [9120] := 48, [9121] := 48, [9122] := 48, [9123] := 48, [9124] := 48, [9125] := 48, [9126] := 44, [9127] := 54, [9128] := 46, [9129] := 48, [9130] := 48, [9131] := 48, [9132] := 48, [9133] := 48, [9134] := 48, [9135] := 48, [9136] := 48, [9137] := 44, [9138] := 55, [9139] := 46, [9140] := 48, [9141] := 48, [9142] := 48, [9143] := 48, [9144] := 48, [9145] := 48, [9146] := 48, [9147] := 48, [9148] := 44, [9149] := 56, [9150] := 46, [9151] := 48, [9152] := 48, [9153] := 48, [9154] := 48, [9155] := 48, [9156] := 48, [9157] := 48, [9158] := 48, [9159] := 44, [9160] := 57, [9161] := 46, [9162] := 48, [9163] := 48, [9164] := 48, [9165] := 48, [9166] := 48, [9167] := 48, [9168] := 48, [9169] := 48, [9170] := 44, [9171] := 49, [9172] := 48, [9173] := 46, [9174] := 48, [9175] := 48, [9176] := 48, [9177] := 48, [9178] := 48, [9179] := 48,
        [9180] := 48, [9181] := 44, [9182] := 49, [9183] := 49, [9184] := 46, [9185] := 48, [9186] := 48, [9187] := 48, [9188] := 48, [9189] := 48, [9190] := 48, [9191] := 48, [9192] := 44, [9193] := 49, [9194] := 50, [9195] := 46, [9196] := 48, [9197] := 48, [9198] := 48, [9199] := 48, [9200] := 48, [9201] := 48, [9202] := 48, [9203] := 44, [9204] := 49, [9205] := 46, [9206] := 48, [9207] := 48, [9208] := 48, [9209] := 48, [9210] := 48, [9211] := 48, [9212] := 48, [9213] := 48, [9214] := 13, [9215] := 10, [9216] := 51, [9217] := 53, [9218] := 56, [9219] := 56, [9220] := 56, [9221] := 44, [9222] := 48, [9223] := 46, [9224] := 48, [9225] := 57, [9226] := 51, [9227] := 53, [9228] := 51, [9229] := 57, [9230] := 57, [9231] := 51, [9232] := 44, [9233] := 50, [9234] := 46, [9235] := 48, [9236] := 48, [9237] := 48, [9238] := 48, [9239] := 48,
        [9240] := 48, [9241] := 48, [9242] := 48, [9243] := 44, [9244] := 53, [9245] := 46, [9246] := 48, [9247] := 48, [9248] := 48, [9249] := 48, [9250] := 48, [9251] := 48, [9252] := 48, [9253] := 48, [9254] := 44, [9255] := 54, [9256] := 46, [9257] := 48, [9258] := 48, [9259] := 48, [9260] := 48, [9261] := 48, [9262] := 48, [9263] := 48, [9264] := 48, [9265] := 44, [9266] := 55, [9267] := 46, [9268] := 48, [9269] := 48, [9270] := 48, [9271] := 48, [9272] := 48, [9273] := 48, [9274] := 48, [9275] := 48, [9276] := 44, [9277] := 56, [9278] := 46, [9279] := 48, [9280] := 48, [9281] := 48, [9282] := 48, [9283] := 48, [9284] := 48, [9285] := 48, [9286] := 48, [9287] := 44, [9288] := 57, [9289] := 46, [9290] := 48, [9291] := 48, [9292] := 48, [9293] := 48, [9294] := 48, [9295] := 48, [9296] := 48, [9297] := 48, [9298] := 44, [9299] := 49,
        [9300] := 48, [9301] := 46, [9302] := 48, [9303] := 48, [9304] := 48, [9305] := 48, [9306] := 48, [9307] := 48, [9308] := 48, [9309] := 44, [9310] := 49, [9311] := 49, [9312] := 46, [9313] := 48, [9314] := 48, [9315] := 48, [9316] := 48, [9317] := 48, [9318] := 48, [9319] := 48, [9320] := 44, [9321] := 49, [9322] := 50, [9323] := 46, [9324] := 48, [9325] := 48, [9326] := 48, [9327] := 48, [9328] := 48, [9329] := 48, [9330] := 48, [9331] := 44, [9332] := 49, [9333] := 46, [9334] := 48, [9335] := 48, [9336] := 48, [9337] := 48, [9338] := 48, [9339] := 48, [9340] := 48, [9341] := 48, [9342] := 13, [9343] := 10, [9344] := 51, [9345] := 53, [9346] := 56, [9347] := 56, [9348] := 56, [9349] := 44, [9350] := 48, [9351] := 46, [9352] := 48, [9353] := 57, [9354] := 51, [9355] := 53, [9356] := 53, [9357] := 49, [9358] := 53, [9359] := 48,
        [9360] := 44, [9361] := 50, [9362] := 46, [9363] := 48, [9364] := 48, [9365] := 48, [9366] := 48, [9367] := 48, [9368] := 48, [9369] := 48, [9370] := 48, [9371] := 44, [9372] := 53, [9373] := 46, [9374] := 48, [9375] := 48, [9376] := 48, [9377] := 48, [9378] := 48, [9379] := 48, [9380] := 48, [9381] := 48, [9382] := 44, [9383] := 54, [9384] := 46, [9385] := 48, [9386] := 48, [9387] := 48, [9388] := 48, [9389] := 48, [9390] := 48, [9391] := 48, [9392] := 48, [9393] := 44, [9394] := 55, [9395] := 46, [9396] := 48, [9397] := 48, [9398] := 48, [9399] := 48, [9400] := 48, [9401] := 48, [9402] := 48, [9403] := 48, [9404] := 44, [9405] := 56, [9406] := 46, [9407] := 48, [9408] := 48, [9409] := 48, [9410] := 48, [9411] := 48, [9412] := 48, [9413] := 48, [9414] := 48, [9415] := 44, [9416] := 57, [9417] := 46, [9418] := 48, [9419] := 48,
        [9420] := 48, [9421] := 48, [9422] := 48, [9423] := 48, [9424] := 48, [9425] := 48, [9426] := 44, [9427] := 49, [9428] := 48, [9429] := 46, [9430] := 48, [9431] := 48, [9432] := 48, [9433] := 48, [9434] := 48, [9435] := 48, [9436] := 48, [9437] := 44, [9438] := 49, [9439] := 49, [9440] := 46, [9441] := 48, [9442] := 48, [9443] := 48, [9444] := 48, [9445] := 48, [9446] := 48, [9447] := 48, [9448] := 44, [9449] := 49, [9450] := 50, [9451] := 46, [9452] := 48, [9453] := 48, [9454] := 48, [9455] := 48, [9456] := 48, [9457] := 48, [9458] := 48, [9459] := 44, [9460] := 49, [9461] := 46, [9462] := 48, [9463] := 48, [9464] := 48, [9465] := 48, [9466] := 48, [9467] := 48, [9468] := 48, [9469] := 48, [9470] := 13, [9471] := 10, [9472] := 51, [9473] := 53, [9474] := 56, [9475] := 56, [9476] := 56, [9477] := 44, [9478] := 48, [9479] := 46,
        [9480] := 48, [9481] := 57, [9482] := 51, [9483] := 53, [9484] := 54, [9485] := 51, [9486] := 48, [9487] := 56, [9488] := 44, [9489] := 50, [9490] := 46, [9491] := 48, [9492] := 48, [9493] := 48, [9494] := 48, [9495] := 48, [9496] := 48, [9497] := 48, [9498] := 48, [9499] := 44, [9500] := 53, [9501] := 46, [9502] := 48, [9503] := 48, [9504] := 48, [9505] := 48, [9506] := 48, [9507] := 48, [9508] := 48, [9509] := 48, [9510] := 44, [9511] := 54, [9512] := 46, [9513] := 48, [9514] := 48, [9515] := 48, [9516] := 48, [9517] := 48, [9518] := 48, [9519] := 48, [9520] := 48, [9521] := 44, [9522] := 55, [9523] := 46, [9524] := 48, [9525] := 48, [9526] := 48, [9527] := 48, [9528] := 48, [9529] := 48, [9530] := 48, [9531] := 48, [9532] := 44, [9533] := 56, [9534] := 46, [9535] := 48, [9536] := 48, [9537] := 48, [9538] := 48, [9539] := 48,
        [9540] := 48, [9541] := 48, [9542] := 48, [9543] := 44, [9544] := 57, [9545] := 46, [9546] := 48, [9547] := 48, [9548] := 48, [9549] := 48, [9550] := 48, [9551] := 48, [9552] := 48, [9553] := 48, [9554] := 44, [9555] := 49, [9556] := 48, [9557] := 46, [9558] := 48, [9559] := 48, [9560] := 48, [9561] := 48, [9562] := 48, [9563] := 48, [9564] := 48, [9565] := 44, [9566] := 49, [9567] := 49, [9568] := 46, [9569] := 48, [9570] := 48, [9571] := 48, [9572] := 48, [9573] := 48, [9574] := 48, [9575] := 48, [9576] := 44, [9577] := 49, [9578] := 50, [9579] := 46, [9580] := 48, [9581] := 48, [9582] := 48, [9583] := 48, [9584] := 48, [9585] := 48, [9586] := 48, [9587] := 44, [9588] := 49, [9589] := 46, [9590] := 48, [9591] := 48, [9592] := 48, [9593] := 48, [9594] := 48, [9595] := 48, [9596] := 48, [9597] := 48, [9598] := 13, [9599] := 10,
        [9600] := 51, [9601] := 53, [9602] := 56, [9603] := 56, [9604] := 56, [9605] := 44, [9606] := 48, [9607] := 46, [9608] := 48, [9609] := 57, [9610] := 51, [9611] := 53, [9612] := 55, [9613] := 52, [9614] := 54, [9615] := 53, [9616] := 44, [9617] := 50, [9618] := 46, [9619] := 48, [9620] := 48, [9621] := 48, [9622] := 48, [9623] := 48, [9624] := 48, [9625] := 48, [9626] := 48, [9627] := 44, [9628] := 53, [9629] := 46, [9630] := 48, [9631] := 48, [9632] := 48, [9633] := 48, [9634] := 48, [9635] := 48, [9636] := 48, [9637] := 48, [9638] := 44, [9639] := 54, [9640] := 46, [9641] := 48, [9642] := 48, [9643] := 48, [9644] := 48, [9645] := 48, [9646] := 48, [9647] := 48, [9648] := 48, [9649] := 44, [9650] := 55, [9651] := 46, [9652] := 48, [9653] := 48, [9654] := 48, [9655] := 48, [9656] := 48, [9657] := 48, [9658] := 48, [9659] := 48,
        [9660] := 44, [9661] := 56, [9662] := 46, [9663] := 48, [9664] := 48, [9665] := 48, [9666] := 48, [9667] := 48, [9668] := 48, [9669] := 48, [9670] := 48, [9671] := 44, [9672] := 57, [9673] := 46, [9674] := 48, [9675] := 48, [9676] := 48, [9677] := 48, [9678] := 48, [9679] := 48, [9680] := 48, [9681] := 48, [9682] := 44, [9683] := 49, [9684] := 48, [9685] := 46, [9686] := 48, [9687] := 48, [9688] := 48, [9689] := 48, [9690] := 48, [9691] := 48, [9692] := 48, [9693] := 44, [9694] := 49, [9695] := 49, [9696] := 46, [9697] := 48, [9698] := 48, [9699] := 48, [9700] := 48, [9701] := 48, [9702] := 48, [9703] := 48, [9704] := 44, [9705] := 49, [9706] := 50, [9707] := 46, [9708] := 48, [9709] := 48, [9710] := 48, [9711] := 48, [9712] := 48, [9713] := 48, [9714] := 48, [9715] := 44, [9716] := 49, [9717] := 46, [9718] := 48, [9719] := 48,
        [9720] := 48, [9721] := 48, [9722] := 48, [9723] := 48, [9724] := 48, [9725] := 48, [9726] := 13, [9727] := 10, [9728] := 51, [9729] := 53, [9730] := 56, [9731] := 56, [9732] := 56, [9733] := 44, [9734] := 48, [9735] := 46, [9736] := 48, [9737] := 57, [9738] := 51, [9739] := 53, [9740] := 56, [9741] := 54, [9742] := 50, [9743] := 52, [9744] := 44, [9745] := 50, [9746] := 46, [9747] := 48, [9748] := 48, [9749] := 48, [9750] := 48, [9751] := 48, [9752] := 48, [9753] := 48, [9754] := 48, [9755] := 44, [9756] := 53, [9757] := 46, [9758] := 48, [9759] := 48, [9760] := 48, [9761] := 48, [9762] := 48, [9763] := 48, [9764] := 48, [9765] := 48, [9766] := 44, [9767] := 54, [9768] := 46, [9769] := 48, [9770] := 48, [9771] := 48, [9772] := 48, [9773] := 48, [9774] := 48, [9775] := 48, [9776] := 48, [9777] := 44, [9778] := 55, [9779] := 46,
        [9780] := 48, [9781] := 48, [9782] := 48, [9783] := 48, [9784] := 48, [9785] := 48, [9786] := 48, [9787] := 48, [9788] := 44, [9789] := 56, [9790] := 46, [9791] := 48, [9792] := 48, [9793] := 48, [9794] := 48, [9795] := 48, [9796] := 48, [9797] := 48, [9798] := 48, [9799] := 44, [9800] := 57, [9801] := 46, [9802] := 48, [9803] := 48, [9804] := 48, [9805] := 48, [9806] := 48, [9807] := 48, [9808] := 48, [9809] := 48, [9810] := 44, [9811] := 49, [9812] := 48, [9813] := 46, [9814] := 48, [9815] := 48, [9816] := 48, [9817] := 48, [9818] := 48, [9819] := 48, [9820] := 48, [9821] := 44, [9822] := 49, [9823] := 49, [9824] := 46, [9825] := 48, [9826] := 48, [9827] := 48, [9828] := 48, [9829] := 48, [9830] := 48, [9831] := 48, [9832] := 44, [9833] := 49, [9834] := 50, [9835] := 46, [9836] := 48, [9837] := 48, [9838] := 48, [9839] := 48,
        [9840] := 48, [9841] := 48, [9842] := 48, [9843] := 44, [9844] := 49, [9845] := 46, [9846] := 48, [9847] := 48, [9848] := 48, [9849] := 48, [9850] := 48, [9851] := 48, [9852] := 48, [9853] := 48, [9854] := 13, [9855] := 10, [9856] := 51, [9857] := 53, [9858] := 56, [9859] := 56, [9860] := 56, [9861] := 44, [9862] := 48, [9863] := 46, [9864] := 48, [9865] := 57, [9866] := 51, [9867] := 53, [9868] := 57, [9869] := 55, [9870] := 56, [9871] := 48, [9872] := 44, [9873] := 50, [9874] := 46, [9875] := 48, [9876] := 48, [9877] := 48, [9878] := 48, [9879] := 48, [9880] := 48, [9881] := 48, [9882] := 48, [9883] := 44, [9884] := 53, [9885] := 46, [9886] := 48, [9887] := 48, [9888] := 48, [9889] := 48, [9890] := 48, [9891] := 48, [9892] := 48, [9893] := 48, [9894] := 44, [9895] := 54, [9896] := 46, [9897] := 48, [9898] := 48, [9899] := 48,
        [9900] := 48, [9901] := 48, [9902] := 48, [9903] := 48, [9904] := 48, [9905] := 44, [9906] := 55, [9907] := 46, [9908] := 48, [9909] := 48, [9910] := 48, [9911] := 48, [9912] := 48, [9913] := 48, [9914] := 48, [9915] := 48, [9916] := 44, [9917] := 56, [9918] := 46, [9919] := 48, [9920] := 48, [9921] := 48, [9922] := 48, [9923] := 48, [9924] := 48, [9925] := 48, [9926] := 48, [9927] := 44, [9928] := 57, [9929] := 46, [9930] := 48, [9931] := 48, [9932] := 48, [9933] := 48, [9934] := 48, [9935] := 48, [9936] := 48, [9937] := 48, [9938] := 44, [9939] := 49, [9940] := 48, [9941] := 46, [9942] := 48, [9943] := 48, [9944] := 48, [9945] := 48, [9946] := 48, [9947] := 48, [9948] := 48, [9949] := 44, [9950] := 49, [9951] := 49, [9952] := 46, [9953] := 48, [9954] := 48, [9955] := 48, [9956] := 48, [9957] := 48, [9958] := 48, [9959] := 48,
        [9960] := 44, [9961] := 49, [9962] := 50, [9963] := 46, [9964] := 48, [9965] := 48, [9966] := 48, [9967] := 48, [9968] := 48, [9969] := 48, [9970] := 48, [9971] := 44, [9972] := 49, [9973] := 46, [9974] := 48, [9975] := 48, [9976] := 48, [9977] := 48, [9978] := 48, [9979] := 48, [9980] := 48, [9981] := 48, [9982] := 13, [9983] := 10, [9984] := 51, [9985] := 53, [9986] := 56, [9987] := 56, [9988] := 56, [9989] := 44, [9990] := 48, [9991] := 46, [9992] := 48, [9993] := 57, [9994] := 51, [9995] := 54, [9996] := 48, [9997] := 57, [9998] := 51, [9999] := 56, [10000] := 44, [10001] := 50, [10002] := 46, [10003] := 48, [10004] := 48, [10005] := 48, [10006] := 48, [10007] := 48, [10008] := 48, [10009] := 48, [10010] := 48, [10011] := 44, [10012] := 53, [10013] := 46, [10014] := 48, [10015] := 48, [10016] := 48, [10017] := 48, [10018] := 48, [10019] := 48,
        [10020] := 48, [10021] := 48, [10022] := 44, [10023] := 54, [10024] := 46, [10025] := 48, [10026] := 48, [10027] := 48, [10028] := 48, [10029] := 48, [10030] := 48, [10031] := 48, [10032] := 48, [10033] := 44, [10034] := 55, [10035] := 46, [10036] := 48, [10037] := 48, [10038] := 48, [10039] := 48, [10040] := 48, [10041] := 48, [10042] := 48, [10043] := 48, [10044] := 44, [10045] := 56, [10046] := 46, [10047] := 48, [10048] := 48, [10049] := 48, [10050] := 48, [10051] := 48, [10052] := 48, [10053] := 48, [10054] := 48, [10055] := 44, [10056] := 57, [10057] := 46, [10058] := 48, [10059] := 48, [10060] := 48, [10061] := 48, [10062] := 48, [10063] := 48, [10064] := 48, [10065] := 48, [10066] := 44, [10067] := 49, [10068] := 48, [10069] := 46, [10070] := 48, [10071] := 48, [10072] := 48, [10073] := 48, [10074] := 48, [10075] := 48, [10076] := 48, [10077] := 44, [10078] := 49, [10079] := 49,
        [10080] := 46, [10081] := 48, [10082] := 48, [10083] := 48, [10084] := 48, [10085] := 48, [10086] := 48, [10087] := 48, [10088] := 44, [10089] := 49, [10090] := 50, [10091] := 46, [10092] := 48, [10093] := 48, [10094] := 48, [10095] := 48, [10096] := 48, [10097] := 48, [10098] := 48, [10099] := 44, [10100] := 49, [10101] := 46, [10102] := 48, [10103] := 48, [10104] := 48, [10105] := 48, [10106] := 48, [10107] := 48, [10108] := 48, [10109] := 48, [10110] := 13, [10111] := 10, [10112] := 49, [10113] := 48, [10114] := 44, [10115] := 54, [10116] := 46, [10117] := 54, [10118] := 54, [10119] := 54, [10120] := 54, [10121] := 54, [10122] := 54, [10123] := 48, [10124] := 51, [10125] := 44, [10126] := 55, [10127] := 46, [10128] := 55, [10129] := 55, [10130] := 55, [10131] := 55, [10132] := 55, [10133] := 55, [10134] := 54, [10135] := 55, [10136] := 44, [10137] := 56, [10138] := 46, [10139] := 56,
        [10140] := 56, [10141] := 56, [10142] := 56, [10143] := 56, [10144] := 57, [10145] := 51, [10146] := 49, [10147] := 44, [10148] := 49, [10149] := 48, [10150] := 46, [10151] := 48, [10152] := 48, [10153] := 48, [10154] := 48, [10155] := 48, [10156] := 48, [10157] := 48, [10158] := 44, [10159] := 48, [10160] := 46, [10161] := 48, [10162] := 13, [10163] := 10, [10164] := 52, [10165] := 49, [10166] := 56, [10167] := 48, [10168] := 51, [10169] := 44, [10170] := 48, [10171] := 46, [10172] := 51, [10173] := 50, [10174] := 53, [10175] := 50, [10176] := 50, [10177] := 57, [10178] := 48, [10179] := 50, [10180] := 44, [10181] := 49, [10182] := 46, [10183] := 49, [10184] := 48, [10185] := 48, [10186] := 48, [10187] := 48, [10188] := 48, [10189] := 48, [10190] := 50, [10191] := 44, [10192] := 50, [10193] := 46, [10194] := 50, [10195] := 50, [10196] := 48, [10197] := 48, [10198] := 48, [10199] := 48,
        [10200] := 48, [10201] := 51, [10202] := 44, [10203] := 51, [10204] := 46, [10205] := 51, [10206] := 51, [10207] := 50, [10208] := 57, [10209] := 57, [10210] := 57, [10211] := 57, [10212] := 52, [10213] := 44, [10214] := 52, [10215] := 46, [10216] := 52, [10217] := 52, [10218] := 52, [10219] := 51, [10220] := 57, [10221] := 57, [10222] := 56, [10223] := 51, [10224] := 44, [10225] := 53, [10226] := 46, [10227] := 53, [10228] := 53, [10229] := 53, [10230] := 53, [10231] := 53, [10232] := 48, [10233] := 49, [10234] := 48, [10235] := 44, [10236] := 54, [10237] := 46, [10238] := 54, [10239] := 54, [10240] := 54, [10241] := 54, [10242] := 54, [10243] := 54, [10244] := 48, [10245] := 51, [10246] := 44, [10247] := 55, [10248] := 46, [10249] := 55, [10250] := 55, [10251] := 55, [10252] := 55, [10253] := 55, [10254] := 55, [10255] := 54, [10256] := 55, [10257] := 44, [10258] := 56, [10259] := 46,
        [10260] := 56, [10261] := 56, [10262] := 56, [10263] := 56, [10264] := 56, [10265] := 57, [10266] := 51, [10267] := 49, [10268] := 44, [10269] := 49, [10270] := 48, [10271] := 46, [10272] := 48, [10273] := 48, [10274] := 48, [10275] := 48, [10276] := 48, [10277] := 48, [10278] := 48, [10279] := 44, [10280] := 48, [10281] := 46, [10282] := 48, [10283] := 13, [10284] := 10, [10285] := 52, [10286] := 49, [10287] := 56, [10288] := 48, [10289] := 51, [10290] := 44, [10291] := 48, [10292] := 46, [10293] := 51, [10294] := 50, [10295] := 53, [10296] := 50, [10297] := 52, [10298] := 48, [10299] := 54, [10300] := 49, [10301] := 44, [10302] := 49, [10303] := 46, [10304] := 49, [10305] := 48, [10306] := 48, [10307] := 48, [10308] := 48, [10309] := 48, [10310] := 48, [10311] := 50, [10312] := 44, [10313] := 50, [10314] := 46, [10315] := 50, [10316] := 50, [10317] := 48, [10318] := 48, [10319] := 48,
        [10320] := 48, [10321] := 48, [10322] := 51, [10323] := 44, [10324] := 51, [10325] := 46, [10326] := 51, [10327] := 51, [10328] := 50, [10329] := 57, [10330] := 57, [10331] := 57, [10332] := 57, [10333] := 52, [10334] := 44, [10335] := 52, [10336] := 46, [10337] := 52, [10338] := 52, [10339] := 52, [10340] := 51, [10341] := 57, [10342] := 57, [10343] := 56, [10344] := 51, [10345] := 44, [10346] := 53, [10347] := 46, [10348] := 53, [10349] := 53, [10350] := 53, [10351] := 53, [10352] := 53, [10353] := 48, [10354] := 49, [10355] := 48, [10356] := 44, [10357] := 54, [10358] := 46, [10359] := 54, [10360] := 54, [10361] := 54, [10362] := 54, [10363] := 54, [10364] := 54, [10365] := 48, [10366] := 51, [10367] := 44, [10368] := 55, [10369] := 46, [10370] := 55, [10371] := 55, [10372] := 55, [10373] := 55, [10374] := 55, [10375] := 55, [10376] := 54, [10377] := 55, [10378] := 44, [10379] := 56,
        [10380] := 46, [10381] := 56, [10382] := 56, [10383] := 56, [10384] := 56, [10385] := 56, [10386] := 57, [10387] := 51, [10388] := 49, [10389] := 44, [10390] := 49, [10391] := 48, [10392] := 46, [10393] := 48, [10394] := 48, [10395] := 48, [10396] := 48, [10397] := 48, [10398] := 48, [10399] := 48, [10400] := 44, [10401] := 48, [10402] := 46, [10403] := 48, [10404] := 13, [10405] := 10, [10406] := 52, [10407] := 49, [10408] := 56, [10409] := 48, [10410] := 51, [10411] := 44, [10412] := 48, [10413] := 46, [10414] := 51, [10415] := 50, [10416] := 53, [10417] := 50, [10418] := 53, [10419] := 50, [10420] := 49, [10421] := 56, [10422] := 44, [10423] := 49, [10424] := 46, [10425] := 49, [10426] := 48, [10427] := 48, [10428] := 48, [10429] := 48, [10430] := 48, [10431] := 48, [10432] := 50, [10433] := 44, [10434] := 50, [10435] := 46, [10436] := 50, [10437] := 50, [10438] := 48, [10439] := 48,
        [10440] := 48, [10441] := 48, [10442] := 48, [10443] := 51, [10444] := 44, [10445] := 51, [10446] := 46, [10447] := 51, [10448] := 51, [10449] := 50, [10450] := 57, [10451] := 57, [10452] := 57, [10453] := 57, [10454] := 52, [10455] := 44, [10456] := 52, [10457] := 46, [10458] := 52, [10459] := 52, [10460] := 52, [10461] := 51, [10462] := 57, [10463] := 57, [10464] := 56, [10465] := 51, [10466] := 44, [10467] := 53, [10468] := 46, [10469] := 53, [10470] := 53, [10471] := 53, [10472] := 53, [10473] := 53, [10474] := 48, [10475] := 49, [10476] := 48, [10477] := 44, [10478] := 54, [10479] := 46, [10480] := 54, [10481] := 54, [10482] := 54, [10483] := 54, [10484] := 54, [10485] := 54, [10486] := 48, [10487] := 51, [10488] := 44, [10489] := 55, [10490] := 46, [10491] := 55, [10492] := 55, [10493] := 55, [10494] := 55, [10495] := 55, [10496] := 55, [10497] := 54, [10498] := 55, [10499] := 44,
        [10500] := 56, [10501] := 46, [10502] := 56, [10503] := 56, [10504] := 56, [10505] := 56, [10506] := 56, [10507] := 57, [10508] := 51, [10509] := 49, [10510] := 44, [10511] := 49, [10512] := 48, [10513] := 46, [10514] := 48, [10515] := 48, [10516] := 48, [10517] := 48, [10518] := 48, [10519] := 48, [10520] := 48, [10521] := 44, [10522] := 48, [10523] := 46, [10524] := 48, [10525] := 13, [10526] := 10, [10527] := 52, [10528] := 49, [10529] := 56, [10530] := 48, [10531] := 51, [10532] := 44, [10533] := 48, [10534] := 46, [10535] := 51, [10536] := 50, [10537] := 53, [10538] := 50, [10539] := 54, [10540] := 51, [10541] := 55, [10542] := 52, [10543] := 44, [10544] := 49, [10545] := 46, [10546] := 49, [10547] := 48, [10548] := 48, [10549] := 48, [10550] := 48, [10551] := 48, [10552] := 48, [10553] := 50, [10554] := 44, [10555] := 50, [10556] := 46, [10557] := 50, [10558] := 50, [10559] := 48,
        [10560] := 48, [10561] := 48, [10562] := 48, [10563] := 48, [10564] := 51, [10565] := 44, [10566] := 51, [10567] := 46, [10568] := 51, [10569] := 51, [10570] := 50, [10571] := 57, [10572] := 57, [10573] := 57, [10574] := 57, [10575] := 52, [10576] := 44, [10577] := 52, [10578] := 46, [10579] := 52, [10580] := 52, [10581] := 52, [10582] := 51, [10583] := 57, [10584] := 57, [10585] := 56, [10586] := 51, [10587] := 44, [10588] := 53, [10589] := 46, [10590] := 53, [10591] := 53, [10592] := 53, [10593] := 53, [10594] := 53, [10595] := 48, [10596] := 49, [10597] := 48, [10598] := 44, [10599] := 54, [10600] := 46, [10601] := 54, [10602] := 54, [10603] := 54, [10604] := 54, [10605] := 54, [10606] := 54, [10607] := 48, [10608] := 51, [10609] := 44, [10610] := 55, [10611] := 46, [10612] := 55, [10613] := 55, [10614] := 55, [10615] := 55, [10616] := 55, [10617] := 55, [10618] := 54, [10619] := 55,
        [10620] := 44, [10621] := 56, [10622] := 46, [10623] := 56, [10624] := 56, [10625] := 56, [10626] := 56, [10627] := 56, [10628] := 57, [10629] := 51, [10630] := 49, [10631] := 44, [10632] := 49, [10633] := 48, [10634] := 46, [10635] := 48, [10636] := 48, [10637] := 48, [10638] := 48, [10639] := 48, [10640] := 48, [10641] := 48, [10642] := 44, [10643] := 48, [10644] := 46, [10645] := 48, [10646] := 13, [10647] := 10, [10648] := 52, [10649] := 49, [10650] := 56, [10651] := 48, [10652] := 51, [10653] := 44, [10654] := 48, [10655] := 46, [10656] := 51, [10657] := 50, [10658] := 53, [10659] := 50, [10660] := 55, [10661] := 53, [10662] := 51, [10663] := 51, [10664] := 44, [10665] := 49, [10666] := 46, [10667] := 49, [10668] := 48, [10669] := 48, [10670] := 48, [10671] := 48, [10672] := 48, [10673] := 48, [10674] := 50, [10675] := 44, [10676] := 50, [10677] := 46, [10678] := 50, [10679] := 50,
        [10680] := 48, [10681] := 48, [10682] := 48, [10683] := 48, [10684] := 48, [10685] := 51, [10686] := 44, [10687] := 51, [10688] := 46, [10689] := 51, [10690] := 51, [10691] := 50, [10692] := 57, [10693] := 57, [10694] := 57, [10695] := 57, [10696] := 52, [10697] := 44, [10698] := 52, [10699] := 46, [10700] := 52, [10701] := 52, [10702] := 52, [10703] := 51, [10704] := 57, [10705] := 57, [10706] := 56, [10707] := 51, [10708] := 44, [10709] := 53, [10710] := 46, [10711] := 53, [10712] := 53, [10713] := 53, [10714] := 53, [10715] := 53, [10716] := 48, [10717] := 49, [10718] := 48, [10719] := 44, [10720] := 54, [10721] := 46, [10722] := 54, [10723] := 54, [10724] := 54, [10725] := 54, [10726] := 54, [10727] := 54, [10728] := 48, [10729] := 51, [10730] := 44, [10731] := 55, [10732] := 46, [10733] := 55, [10734] := 55, [10735] := 55, [10736] := 55, [10737] := 55, [10738] := 55, [10739] := 54,
        [10740] := 55, [10741] := 44, [10742] := 56, [10743] := 46, [10744] := 56, [10745] := 56, [10746] := 56, [10747] := 56, [10748] := 56, [10749] := 57, [10750] := 51, [10751] := 49, [10752] := 44, [10753] := 49, [10754] := 48, [10755] := 46, [10756] := 48, [10757] := 48, [10758] := 48, [10759] := 48, [10760] := 48, [10761] := 48, [10762] := 48, [10763] := 44, [10764] := 48, [10765] := 46, [10766] := 48, [10767] := 13, [10768] := 10, [10769] := 52, [10770] := 49, [10771] := 56, [10772] := 48, [10773] := 51, [10774] := 44, [10775] := 48, [10776] := 46, [10777] := 51, [10778] := 50, [10779] := 53, [10780] := 50, [10781] := 56, [10782] := 54, [10783] := 57, [10784] := 48, [10785] := 44, [10786] := 49, [10787] := 46, [10788] := 49, [10789] := 48, [10790] := 48, [10791] := 48, [10792] := 48, [10793] := 48, [10794] := 48, [10795] := 50, [10796] := 44, [10797] := 50, [10798] := 46, [10799] := 50,
        [10800] := 50, [10801] := 48, [10802] := 48, [10803] := 48, [10804] := 48, [10805] := 48, [10806] := 51, [10807] := 44, [10808] := 51, [10809] := 46, [10810] := 51, [10811] := 51, [10812] := 50, [10813] := 57, [10814] := 57, [10815] := 57, [10816] := 57, [10817] := 52, [10818] := 44, [10819] := 52, [10820] := 46, [10821] := 52, [10822] := 52, [10823] := 52, [10824] := 51, [10825] := 57, [10826] := 57, [10827] := 56, [10828] := 51, [10829] := 44, [10830] := 53, [10831] := 46, [10832] := 53, [10833] := 53, [10834] := 53, [10835] := 53, [10836] := 53, [10837] := 48, [10838] := 49, [10839] := 48, [10840] := 44, [10841] := 54, [10842] := 46, [10843] := 54, [10844] := 54, [10845] := 54, [10846] := 54, [10847] := 54, [10848] := 54, [10849] := 48, [10850] := 51, [10851] := 44, [10852] := 55, [10853] := 46, [10854] := 55, [10855] := 55, [10856] := 55, [10857] := 55, [10858] := 55, [10859] := 55,
        [10860] := 54, [10861] := 55, [10862] := 44, [10863] := 56, [10864] := 46, [10865] := 56, [10866] := 56, [10867] := 56, [10868] := 56, [10869] := 56, [10870] := 57, [10871] := 51, [10872] := 49, [10873] := 44, [10874] := 49, [10875] := 48, [10876] := 46, [10877] := 48, [10878] := 48, [10879] := 48, [10880] := 48, [10881] := 48, [10882] := 48, [10883] := 48, [10884] := 44, [10885] := 48, [10886] := 46, [10887] := 48, [10888] := 13, [10889] := 10, [10890] := 52, [10891] := 49, [10892] := 56, [10893] := 48, [10894] := 51, [10895] := 44, [10896] := 48, [10897] := 46, [10898] := 51, [10899] := 50, [10900] := 53, [10901] := 50, [10902] := 57, [10903] := 56, [10904] := 52, [10905] := 54, [10906] := 44, [10907] := 49, [10908] := 46, [10909] := 49, [10910] := 48, [10911] := 48, [10912] := 48, [10913] := 48, [10914] := 48, [10915] := 48, [10916] := 50, [10917] := 44, [10918] := 50, [10919] := 46,
        [10920] := 50, [10921] := 50, [10922] := 48, [10923] := 48, [10924] := 48, [10925] := 48, [10926] := 48, [10927] := 51, [10928] := 44, [10929] := 51, [10930] := 46, [10931] := 51, [10932] := 51, [10933] := 50, [10934] := 57, [10935] := 57, [10936] := 57, [10937] := 57, [10938] := 52, [10939] := 44, [10940] := 52, [10941] := 46, [10942] := 52, [10943] := 52, [10944] := 52, [10945] := 51, [10946] := 57, [10947] := 57, [10948] := 56, [10949] := 51, [10950] := 44, [10951] := 53, [10952] := 46, [10953] := 53, [10954] := 53, [10955] := 53, [10956] := 53, [10957] := 53, [10958] := 48, [10959] := 49, [10960] := 48, [10961] := 44, [10962] := 54, [10963] := 46, [10964] := 54, [10965] := 54, [10966] := 54, [10967] := 54, [10968] := 54, [10969] := 54, [10970] := 48, [10971] := 51, [10972] := 44, [10973] := 55, [10974] := 46, [10975] := 55, [10976] := 55, [10977] := 55, [10978] := 55, [10979] := 55,
        [10980] := 55, [10981] := 54, [10982] := 55, [10983] := 44, [10984] := 56, [10985] := 46, [10986] := 56, [10987] := 56, [10988] := 56, [10989] := 56, [10990] := 56, [10991] := 57, [10992] := 51, [10993] := 49, [10994] := 44, [10995] := 49, [10996] := 48, [10997] := 46, [10998] := 48, [10999] := 48);
   CF0x3MSG : MESSAGE;   // detect card
        MessageParameters(ServiceCode := 16#0003, LocalElement := CF_data[0], DestinationTag := CF_data[10], ...)
   CF0x4fMSG : MESSAGE;   // read from file
        MessageParameters(ServiceCode := 16#004f, LocalElement := CF_data[0], DestinationTag := CF_data[20], ...)
   CF0x50MSG : MESSAGE;   // write to file
        MessageParameters(ServiceCode := 16#0050, LocalElement := CF_data[0], DestinationTag := CF_data[500], ...)
   CF0x52MSG : MESSAGE;   // file open
        MessageParameters(ServiceCode := 16#0052, LocalElement := CF_data[0], DestinationTag := CF_data[400], ...)
   CF0x53MSG : MESSAGE;   // set file pointer
        MessageParameters(ServiceCode := 16#0053, LocalElement := CF_data[0], DestinationTag := CF_data[100], ...)
   CF0x54MSG : MESSAGE;   // file close
        MessageParameters(ServiceCode := 16#0054, LocalElement := CF_data[0], DestinationTag := CF_data[100], ...)
   CF0x55MSG : MESSAGE;   // delete file
        MessageParameters(ServiceCode := 16#0055, LocalElement := CF_data[0], DestinationTag := CF_data[400], ...)
   CF0x56MSG : MESSAGE;   // create directory
        MessageParameters(ServiceCode := 16#0056, LocalElement := CF_data[0], DestinationTag := CF_data[400], ...)
   CF0x57MSG : MESSAGE;   // rename/move file
        MessageParameters(ServiceCode := 16#0057, LocalElement := CF_data[0], DestinationTag := CF_data[400], ...)
   CF0x58MSG : MESSAGE;   // Find first file
        MessageParameters(ServiceCode := 16#0058, LocalElement := CF_data[0], DestinationTag := CF_data[100], ...)
   CF0x59MSG : MESSAGE;   // Find next file
        MessageParameters(ServiceCode := 16#0059, LocalElement := CF_data[0], DestinationTag := CF_data[100], ...)
   CF0x5aMSG : MESSAGE;   // Find close
        MessageParameters(ServiceCode := 16#005a, LocalElement := CF_data[0], DestinationTag := CF_data[100], ...)
   CF_data : SINT[512] := ([4] := -120, [5] := 1, [6] := 48, [7] := 48, [8] := 48, [9] := 48, [10] := 48, [11] := 48, [12] := 13, [13] := 10, [14] := 51, [15] := 53, [16] := 56, [17] := 56, [18] := 56, [19] := 44, [20] := 48, [21] := 46, [22] := 48, [23] := 57, [24] := 51, [25] := 53, [26] := 56, [27] := 54, [28] := 50, [29] := 52, [30] := 44, [31] := 50, [32] := 46, [33] := 48, [34] := 48, [35] := 48, [36] := 48, [37] := 48, [38] := 48, [39] := 48, [40] := 48, [41] := 44, [42] := 53, [43] := 46, [44] := 48, [45] := 48, [46] := 48, [47] := 48, [48] := 48, [49] := 48, [50] := 48, [51] := 48, [52] := 44, [53] := 54, [54] := 46, [55] := 48, [56] := 48, [57] := 48, [58] := 48, [59] := 48, [60] := 48, [61] := 48, [62] := 48, [63] := 44,
        [64] := 55, [65] := 46, [66] := 48, [67] := 48, [68] := 48, [69] := 48, [70] := 48, [71] := 48, [72] := 48, [73] := 48, [74] := 44, [75] := 56, [76] := 46, [77] := 48, [78] := 48, [79] := 48, [80] := 48, [81] := 48, [82] := 48, [83] := 48, [84] := 48, [85] := 44, [86] := 57, [87] := 46, [88] := 48, [89] := 48, [90] := 48, [91] := 48, [92] := 48, [93] := 48, [94] := 48, [95] := 48, [96] := 44, [97] := 49, [98] := 48, [99] := 46, [100] := 48, [101] := 48, [102] := 48, [103] := 48, [104] := 48, [105] := 48, [106] := 48, [107] := 44, [108] := 49, [109] := 49, [110] := 46, [111] := 48, [112] := 48, [113] := 48, [114] := 48, [115] := 48, [116] := 48, [117] := 48, [118] := 44, [119] := 49, [120] := 50, [121] := 46, [122] := 48, [123] := 48,
        [124] := 48, [125] := 48, [126] := 48, [127] := 48, [128] := 48, [129] := 44, [130] := 49, [131] := 46, [132] := 48, [133] := 48, [134] := 48, [135] := 48, [136] := 48, [137] := 48, [138] := 48, [139] := 48, [140] := 13, [141] := 10, [142] := 51, [143] := 53, [144] := 56, [145] := 56, [146] := 56, [147] := 44, [148] := 48, [149] := 46, [150] := 48, [151] := 57, [152] := 51, [153] := 53, [154] := 57, [155] := 55, [156] := 56, [157] := 48, [158] := 44, [159] := 50, [160] := 46, [161] := 48, [162] := 48, [163] := 48, [164] := 48, [165] := 48, [166] := 48, [167] := 48, [168] := 48, [169] := 44, [170] := 53, [171] := 46, [172] := 48, [173] := 48, [174] := 48, [175] := 48, [176] := 48, [177] := 48, [178] := 48, [179] := 48, [180] := 44, [181] := 54, [182] := 46, [183] := 48,
        [184] := 48, [185] := 48, [186] := 48, [187] := 48, [188] := 48, [189] := 48, [190] := 48, [191] := 44, [192] := 55, [193] := 46, [194] := 48, [195] := 48, [196] := 48, [197] := 48, [198] := 48, [199] := 48, [200] := 48, [201] := 48, [202] := 44, [203] := 56, [204] := 46, [205] := 48, [206] := 48, [207] := 48, [208] := 48, [209] := 48, [210] := 48, [211] := 48, [212] := 48, [213] := 44, [214] := 57, [215] := 46, [216] := 48, [217] := 48, [218] := 48, [219] := 48, [220] := 48, [221] := 48, [222] := 48, [223] := 48, [224] := 44, [225] := 49, [226] := 48, [227] := 46, [228] := 48, [229] := 48, [230] := 48, [231] := 48, [232] := 48, [233] := 48, [234] := 48, [235] := 44, [236] := 49, [237] := 49, [238] := 46, [239] := 48, [240] := 48, [241] := 48, [242] := 48, [243] := 48,
        [244] := 48, [245] := 48, [246] := 44, [247] := 49, [248] := 50, [249] := 46, [250] := 48, [251] := 48, [252] := 48, [253] := 48, [254] := 48, [255] := 48, [256] := 48, [257] := 44, [258] := 49, [259] := 46, [260] := 48, [261] := 48, [262] := 48, [263] := 48, [264] := 48, [265] := 48, [266] := 48, [267] := 48, [268] := 13, [269] := 10, [270] := 51, [271] := 53, [272] := 56, [273] := 56, [274] := 56, [275] := 44, [276] := 48, [277] := 46, [278] := 48, [279] := 57, [280] := 51, [281] := 54, [282] := 48, [283] := 57, [284] := 51, [285] := 56, [286] := 44, [287] := 50, [288] := 46, [289] := 48, [290] := 48, [291] := 48, [292] := 48, [293] := 48, [294] := 48, [295] := 48, [296] := 48, [297] := 44, [298] := 53, [299] := 46, [300] := 48, [301] := 48, [302] := 48, [303] := 48,
        [304] := 48, [305] := 48, [306] := 48, [307] := 48, [308] := 44, [309] := 54, [310] := 46, [311] := 48, [312] := 48, [313] := 48, [314] := 48, [315] := 48, [316] := 48, [317] := 48, [318] := 48, [319] := 44, [320] := 55, [321] := 46, [322] := 48, [323] := 48, [324] := 48, [325] := 48, [326] := 48, [327] := 48, [328] := 48, [329] := 48, [330] := 44, [331] := 56, [332] := 46, [333] := 48, [334] := 48, [335] := 48, [336] := 48, [337] := 48, [338] := 48, [339] := 48, [340] := 48, [341] := 44, [342] := 57, [343] := 46, [344] := 48, [345] := 48, [346] := 48, [347] := 48, [348] := 48, [349] := 48, [350] := 48, [351] := 48, [352] := 44, [353] := 49, [354] := 48, [355] := 46, [356] := 48, [357] := 48, [358] := 48, [359] := 48, [360] := 48, [361] := 48, [362] := 48, [363] := 44,
        [364] := 49, [365] := 49, [366] := 46, [367] := 48, [368] := 48, [369] := 48, [370] := 48, [371] := 48, [372] := 48, [373] := 48, [374] := 44, [375] := 49, [376] := 50, [377] := 46, [378] := 48, [379] := 48, [380] := 48, [381] := 48, [382] := 48, [383] := 48, [384] := 48, [385] := 44, [386] := 49, [387] := 46, [388] := 48, [389] := 48, [390] := 48, [391] := 48, [392] := 48, [393] := 48, [394] := 48, [395] := 48, [396] := 13, [397] := 10, [398] := 48, [399] := 48, [400] := 48, [401] := 48, [402] := 48, [403] := 48, [404] := 48, [405] := 48, [406] := 44, [407] := 56, [408] := 46, [409] := 48, [410] := 48, [411] := 48, [412] := 48, [413] := 48, [414] := 48, [415] := 48, [416] := 48, [417] := 44, [418] := 57, [419] := 46, [420] := 48, [421] := 48, [422] := 48, [423] := 48,
        [424] := 48, [425] := 48, [426] := 48, [427] := 48, [428] := 44, [429] := 49, [430] := 48, [431] := 46, [432] := 48, [433] := 48, [434] := 48, [435] := 48, [436] := 48, [437] := 48, [438] := 48, [439] := 44, [440] := 49, [441] := 49, [442] := 46, [443] := 48, [444] := 48, [445] := 48, [446] := 48, [447] := 48, [448] := 48, [449] := 48, [450] := 44, [451] := 49, [452] := 50, [453] := 46, [454] := 48, [455] := 48, [456] := 48, [457] := 48, [458] := 48, [459] := 48, [460] := 48, [461] := 44, [462] := 49, [463] := 46, [464] := 48, [465] := 48, [466] := 116, [467] := 117, [468] := 118, [469] := 119, [470] := 120, [471] := 121, [472] := 97, [473] := 98, [474] := 99, [475] := 100, [476] := 101, [477] := 102, [478] := 103, [479] := 104, [480] := 105, [481] := 106, [482] := 102, [483] := 103,
        [484] := 104, [485] := 105, [486] := 106, [487] := 107, [488] := 108, [489] := 109, [490] := 110, [491] := 111, [492] := 112, [493] := 113, [494] := 114, [495] := 115, [496] := 116, [497] := 117, [498] := 118, [499] := 88, [500] := -120, [501] := 1);
   CF_RW_functions : CF_functions := (index := 10, REQ_length := 4992, DN_length := 4992, result := 25216, name := 'Log_1998_04_03_02_11.csv', data[0] := 48, data[1] := 48, data[2] := 48, data[3] := 48, data[4] := 48, data[5] := 48, data[6] := 13, data[7] := 10, data[8] := 51, data[9] := 53, data[10] := 56, data[11] := 56, data[12] := 56, data[13] := 44, data[14] := 48, data[15] := 46, data[16] := 48, data[17] := 57, data[18] := 51, data[19] := 53, data[20] := 56, data[21] := 54, data[22] := 50, data[23] := 52, data[24] := 44, data[25] := 50, data[26] := 46, data[27] := 48, data[28] := 48, data[29] := 48, data[30] := 48, data[31] := 48, data[32] := 48, data[33] := 48, data[34] := 48, data[35] := 44, data[36] := 53, data[37] := 46, data[38] := 48, data[39] := 48, data[40] := 48, data[41] := 48, data[42] := 48, data[43] := 48, data[44] := 48, data[45] := 48, data[46] := 44, data[47] := 54, data[48] := 46, data[49] := 48, data[50] := 48, data[51] := 48, data[52] := 48, data[53] := 48, data[54] := 48,
        data[55] := 48, data[56] := 48, data[57] := 44, data[58] := 55, data[59] := 46, data[60] := 48, data[61] := 48, data[62] := 48, data[63] := 48, data[64] := 48, data[65] := 48, data[66] := 48, data[67] := 48, data[68] := 44, data[69] := 56, data[70] := 46, data[71] := 48, data[72] := 48, data[73] := 48, data[74] := 48, data[75] := 48, data[76] := 48, data[77] := 48, data[78] := 48, data[79] := 44, data[80] := 57, data[81] := 46, data[82] := 48, data[83] := 48, data[84] := 48, data[85] := 48, data[86] := 48, data[87] := 48, data[88] := 48, data[89] := 48, data[90] := 44, data[91] := 49, data[92] := 48, data[93] := 46, data[94] := 48, data[95] := 48, data[96] := 48, data[97] := 48, data[98] := 48, data[99] := 48, data[100] := 48, data[101] := 44, data[102] := 49, data[103] := 49, data[104] := 46, data[105] := 48, data[106] := 48, data[107] := 48, data[108] := 48, data[109] := 48, data[110] := 48, data[111] := 48, data[112] := 44, data[113] := 49, data[114] := 50,
        data[115] := 46, data[116] := 48, data[117] := 48, data[118] := 48, data[119] := 48, data[120] := 48, data[121] := 48, data[122] := 48, data[123] := 44, data[124] := 49, data[125] := 46, data[126] := 48, data[127] := 48, data[128] := 48, data[129] := 48, data[130] := 48, data[131] := 48, data[132] := 48, data[133] := 48, data[134] := 13, data[135] := 10, data[136] := 51, data[137] := 53, data[138] := 56, data[139] := 56, data[140] := 56, data[141] := 44, data[142] := 48, data[143] := 46, data[144] := 48, data[145] := 57, data[146] := 51, data[147] := 53, data[148] := 57, data[149] := 55, data[150] := 56, data[151] := 48, data[152] := 44, data[153] := 50, data[154] := 46, data[155] := 48, data[156] := 48, data[157] := 48, data[158] := 48, data[159] := 48, data[160] := 48, data[161] := 48, data[162] := 48, data[163] := 44, data[164] := 53, data[165] := 46, data[166] := 48, data[167] := 48, data[168] := 48, data[169] := 48, data[170] := 48, data[171] := 48, data[172] := 48, data[173] := 48, data[174] := 44,
        data[175] := 54, data[176] := 46, data[177] := 48, data[178] := 48, data[179] := 48, data[180] := 48, data[181] := 48, data[182] := 48, data[183] := 48, data[184] := 48, data[185] := 44, data[186] := 55, data[187] := 46, data[188] := 48, data[189] := 48, data[190] := 48, data[191] := 48, data[192] := 48, data[193] := 48, data[194] := 48, data[195] := 48, data[196] := 44, data[197] := 56, data[198] := 46, data[199] := 48, data[200] := 48, data[201] := 48, data[202] := 48, data[203] := 48, data[204] := 48, data[205] := 48, data[206] := 48, data[207] := 44, data[208] := 57, data[209] := 46, data[210] := 48, data[211] := 48, data[212] := 48, data[213] := 48, data[214] := 48, data[215] := 48, data[216] := 48, data[217] := 48, data[218] := 44, data[219] := 49, data[220] := 48, data[221] := 46, data[222] := 48, data[223] := 48, data[224] := 48, data[225] := 48, data[226] := 48, data[227] := 48, data[228] := 48, data[229] := 44, data[230] := 49, data[231] := 49, data[232] := 46, data[233] := 48, data[234] := 48,
        data[235] := 48, data[236] := 48, data[237] := 48, data[238] := 48, data[239] := 48, data[240] := 44, data[241] := 49, data[242] := 50, data[243] := 46, data[244] := 48, data[245] := 48, data[246] := 48, data[247] := 48, data[248] := 48, data[249] := 48, data[250] := 48, data[251] := 44, data[252] := 49, data[253] := 46, data[254] := 48, data[255] := 48, data[256] := 48, data[257] := 48, data[258] := 48, data[259] := 48, data[260] := 48, data[261] := 48, data[262] := 13, data[263] := 10, data[264] := 51, data[265] := 53, data[266] := 56, data[267] := 56, data[268] := 56, data[269] := 44, data[270] := 48, data[271] := 46, data[272] := 48, data[273] := 57, data[274] := 51, data[275] := 54, data[276] := 48, data[277] := 57, data[278] := 51, data[279] := 56, data[280] := 44, data[281] := 50, data[282] := 46, data[283] := 48, data[284] := 48, data[285] := 48, data[286] := 48, data[287] := 48, data[288] := 48, data[289] := 48, data[290] := 48, data[291] := 44, data[292] := 53, data[293] := 46, data[294] := 48,
        data[295] := 48, data[296] := 48, data[297] := 48, data[298] := 48, data[299] := 48, data[300] := 48, data[301] := 48, data[302] := 44, data[303] := 54, data[304] := 46, data[305] := 48, data[306] := 48, data[307] := 48, data[308] := 48, data[309] := 48, data[310] := 48, data[311] := 48, data[312] := 48, data[313] := 44, data[314] := 55, data[315] := 46, data[316] := 48, data[317] := 48, data[318] := 48, data[319] := 48, data[320] := 48, data[321] := 48, data[322] := 48, data[323] := 48, data[324] := 44, data[325] := 56, data[326] := 46, data[327] := 48, data[328] := 48, data[329] := 48, data[330] := 48, data[331] := 48, data[332] := 48, data[333] := 48, data[334] := 48, data[335] := 44, data[336] := 57, data[337] := 46, data[338] := 48, data[339] := 48, data[340] := 48, data[341] := 48, data[342] := 48, data[343] := 48, data[344] := 48, data[345] := 48, data[346] := 44, data[347] := 49, data[348] := 48, data[349] := 46, data[350] := 48, data[351] := 48, data[352] := 48, data[353] := 48, data[354] := 48,
        data[355] := 48, data[356] := 48, data[357] := 44, data[358] := 49, data[359] := 49, data[360] := 46, data[361] := 48, data[362] := 48, data[363] := 48, data[364] := 48, data[365] := 48, data[366] := 48, data[367] := 48, data[368] := 44, data[369] := 49, data[370] := 50, data[371] := 46, data[372] := 48, data[373] := 48, data[374] := 48, data[375] := 48, data[376] := 48, data[377] := 48, data[378] := 48, data[379] := 44, data[380] := 49, data[381] := 46, data[382] := 48, data[383] := 48, data[384] := 48, data[385] := 48, data[386] := 48, data[387] := 48, data[388] := 48, data[389] := 48, data[390] := 13, data[391] := 10, data[392] := 48, data[393] := 48, data[394] := 48, data[395] := 48, data[396] := 48, data[397] := 48, data[398] := 48, data[399] := 48, data[400] := 44, data[401] := 56, data[402] := 46, data[403] := 48, data[404] := 48, data[405] := 48, data[406] := 48, data[407] := 48, data[408] := 48, data[409] := 48, data[410] := 48, data[411] := 44, data[412] := 57, data[413] := 46, data[414] := 48,
        data[415] := 48, data[416] := 48, data[417] := 48, data[418] := 48, data[419] := 48, data[420] := 48, data[421] := 48, data[422] := 44, data[423] := 49, data[424] := 48, data[425] := 46, data[426] := 48, data[427] := 48, data[428] := 48, data[429] := 48, data[430] := 48, data[431] := 48, data[432] := 48, data[433] := 44, data[434] := 49, data[435] := 49, data[436] := 46, data[437] := 48, data[438] := 48, data[439] := 48, data[440] := 48, data[441] := 48, data[442] := 48, data[443] := 48, data[444] := 44, data[445] := 49, data[446] := 50, data[447] := 46, data[448] := 48, data[449] := 48, data[450] := 48, data[451] := 48, data[452] := 48, data[453] := 48, data[454] := 48, data[455] := 44, data[456] := 49, data[457] := 46, data[458] := 48, data[459] := 48, strings[0] := 'Log_1998_03_31_05_28.csv', strings[1] := 'Log_1998_03_31_06_01.csv', strings[2] := 'Log_1998_03_31_06_34.csv', strings[3] := 'Log_1998_03_31_07_09.csv', strings[4] := 'Log_1998_04_01_06_32.csv', strings[5] := 'Log_1998_04_01_07_05.csv', strings[6] := 'Log_1998_04_01_07_38.csv', strings[7] := 'Log_1998_04_01_08_11.csv', strings[8] := 'Log_1998_04_01_08_44.csv', strings[9] := 'Log_1998_04_01_09_17.csv', strings[10] := 'Log_1998_04_01_09_50.csv', strings[11] := 'Log_1998_04_02_01_05.csv', strings[12] := 'Log_1998_04_02_01_37.csv', strings[13] := 'Log_1998_04_02_02_15.csv', strings[14] := 'Log_1998_04_02_02_48.csv',
        strings[15] := 'Log_1998_04_02_03_21.csv', strings[16] := 'Log_1998_04_02_03_54.csv', strings[17] := 'Log_1998_04_02_04_27.csv', strings[18] := 'Log_1998_04_02_05_00.csv', strings[19] := 'Log_1998_04_02_05_33.csv', strings[20] := 'Log_1998_04_02_06_06.csv', strings[21] := 'Log_1998_04_02_06_39.csv', strings[22] := 'Log_1998_04_02_07_12.csv', strings[23] := 'Log_1998_04_02_07_44.csv', strings[24] := 'Log_1998_04_02_08_17.csv', strings[25] := 'Log_1998_04_02_08_50.csv', strings[26] := 'Log_1998_03_11_09_14.csv', strings[27] := 'Log_1998_03_11_09_47.csv', strings[28] := 'Log_1998_03_26_02_51.csv', strings[29] := 'Log_1998_03_30_04_14.csv', strings[30] := 'Log_1998_03_30_04_47.csv', strings[31] := 'Log_1998_03_30_05_20.csv', strings[32] := 'Log_1998_03_30_05_53.csv', strings[33] := 'Log_1998_03_30_06_26.csv', strings[34] := 'Log_1998_03_30_06_59.csv', strings[35] := 'Log_1998_03_30_07_32.csv', strings[36] := 'Log_1998_03_30_08_05.csv', strings[37] := 'Log_1998_03_30_08_38.csv', strings[38] := 'Log_1998_03_30_09_10.csv', strings[39] := 'Log_1998_03_30_09_43.csv', strings[40] := 'Log_1998_03_30_10_16.csv', strings[41] := 'Log_1998_03_30_10_49.csv', strings[42] := 'Log_1998_03_30_11_22.csv', strings[43] := 'Log_1998_03_30_11_55.csv', strings[44] := 'Log_1998_03_30_12_28.csv', strings[45] := 'Log_1998_03_30_13_01.csv', strings[46] := 'Log_1998_03_30_13_34.csv', strings[47] := 'Log_1998_03_30_14_07.csv', strings[48] := 'Log_1998_03_30_14_40.csv', strings[49] := 'Log_1998_03_30_15_13.csv', strings[50] := 'Log_1998_03_30_15_45.csv', strings[51] := 'Log_1998_03_30_16_18.csv', strings[52] := 'Log_1998_03_30_16_51.csv', strings[53] := 'Log_1998_03_30_17_24.csv', strings[54] := 'Log_1998_03_30_17_57.csv', strings[55] := 'Log_1998_03_30_18_30.csv', strings[56] := 'Log_1998_03_30_19_03.csv', strings[57] := 'Log_1998_03_30_19_36.csv', strings[58] := 'Log_1998_03_30_20_09.csv', strings[59] := 'Log_1998_03_30_20_42.csv', strings[60] := 'Log_1998_03_30_21_15.csv', strings[61] := 'Log_1998_03_30_21_48.csv', strings[62] := 'Log_1998_03_30_22_20.csv', strings[63] := 'Log_1998_03_30_22_53.csv', strings[64] := 'Log_1998_03_30_23_26.csv', strings[65] := 'Log_1998_03_30_23_59.csv', strings[66] := 'Log_1998_03_31_00_32.csv', strings[67] := 'Log_1998_03_31_01_05.csv', strings[68] := 'Log_1998_03_31_01_38.csv', strings[69] := 'Log_1998_03_31_02_11.csv', strings[70] := 'Log_1998_03_31_02_44.csv', strings[71] := 'Log_1998_03_31_03_17.csv', strings[72] := 'Log_1998_03_31_03_50.csv', strings[73] := 'Log_1998_03_31_04_23.csv', strings[74] := 'Log_1998_03_31_04_55.csv');
   counters : COUNTER[20];
        [0]   // C indice Dinagrama
   DATE_TIME_SET_TO_PLC : DINT[7];
        [0]   // YEAR
        [1]   // MONTH
        [2]   // DAY
        [3]   // HOUR
        [4]   // MINUTE
        [5]   // SECONDS
        [6]   // MILISECONDS
   manual_log_trigger : BOOL;
   ONS_001 : BOOL;
   PLC_STATUS : INT;
   Proximetro : BOOL := 1;
   SET_TIME : BOOL;
   SrcData : REAL[10] := ([0] := 2.0, [1] := 5.0, [2] := 6.0, [3] := 7.0, [4] := 8.0, [5] := 9.0, [6] := 10.0, [7] := 11.0, [8] := 12.0, [9] := 1.0);
   SWC : SWC := (comand.referencia := 1440.0, comand.direction := 1, dinagrama.indiceAux := 177, dinagrama.indice := 177, dinagrama.PotenciaC := -5.9576063, dinagrama.Potencia := 5.9449345e-37, dinagrama.numeroMuestras := 280, dinagrama.tiempoMuestreo := 31, dinagrama.tiempoPausa := 196, dinagrama.proximetro := 1, dinagrama.Posicion := 4.63953, dinagrama.Carga := 9.607954, dinagrama.confPos.ValorMinAmp := 16.750578, dinagrama.confCarga.ValorMinAmp := 15.609078, dinagrama.confPot.ValorMinAmp := 3.2056525, entradasDigitales := 3, salidasDigitales := 1, entradasAnalogas[0] := 3.2056525, entradasAnalogas[1] := 8.910149, entradasAnalogas[2] := 4.0510225, entradasAnalogas[3] := 4.0120053, ABBRead.Logic_Status_Word.Ready := 1, ABBRead.Logic_Status_Word.RemoteRef := 1, ABBRead.Logic_Status_Word.RemoteCrtl := 1, ABBRead.RPM_Referencia := 1440, ABBRead.Output_Power := 5.9449345e-37, ABBRead.BusDC := 678.2, ABBRead.Latest_Fault := 13185, etheWrite.Enabled := 1, etheWrite.ERR := 1, etheWrite.Value := 1, etheWrite.Instance := 99, etheWrite.Atribute := 13, etheRead.Value := 6000, etheRead.instance := 99, etheRead.atribute := 7);
   Timmers : TIMER[10] := ([0].PRE := 31, [1].PRE := 196000, [2].PRE := 500, [3].PRE := 200, [4].PRE := 10000);
        [0]   // tMuestreo
        [1]   // tPausa
        [2]   // reset del done write ethet
        [3]   // reset del done read eth
        [4]   // reset de la flag de arranque
END_VAR
